   1:L PR[91] R[100]mm/sec CNT100;
   1:  PR[GP1:91,1] = PR[GP1:90,1] + -9.731;
   1:  PR[GP1:91,2] = PR[GP1:90,2] + -19.445;
   1:L PR[91] R[100]mm/sec CNT100;
   1:  PR[GP1:91,1] = PR[GP1:90,1] + -5.449;
   1:  PR[GP1:91,2] = PR[GP1:90,2] + -10.889;
   1:L PR[91] R[100]mm/sec CNT100;
   1:  PR[GP1:91,1] = PR[GP1:90,1] + -4.653;
   1:  PR[GP1:91,2] = PR[GP1:90,2] + -8.576;
   1:L PR[91] R[100]mm/sec CNT100;
   1:  PR[GP1:91,1] = PR[GP1:90,1] + -3.640;
   1:  PR[GP1:91,2] = PR[GP1:90,2] + -7.457;
   1:L PR[91] R[100]mm/sec CNT100;
   1:  PR[GP1:91,1] = PR[GP1:90,1] + -3.365;
   1:  PR[GP1:91,2] = PR[GP1:90,2] + -7.289;
   1:L PR[91] R[100]mm/sec CNT100;
   1:  PR[GP1:91,1] = PR[GP1:90,1] + -1.883;
   1:  PR[GP1:91,2] = PR[GP1:90,2] + -5.517;
   1:L PR[91] R[100]mm/sec CNT100;
   1:  PR[GP1:91,1] = PR[GP1:90,1] + 0.854;
   1:  PR[GP1:91,2] = PR[GP1:90,2] + -5.728;
   1:L PR[91] R[100]mm/sec CNT100;
   1:  PR[GP1:91,1] = PR[GP1:90,1] + 0.970;
   1:  PR[GP1:91,2] = PR[GP1:90,2] + -5.821;
   1:L PR[91] R[100]mm/sec CNT100;
   1:  PR[GP1:91,1] = PR[GP1:90,1] + 2.632;
   1:  PR[GP1:91,2] = PR[GP1:90,2] + -5.804;
   1:L PR[91] R[100]mm/sec CNT100;
   1:  PR[GP1:91,1] = PR[GP1:90,1] + 3.827;
   1:  PR[GP1:91,2] = PR[GP1:90,2] + -8.079;
   1:L PR[91] R[100]mm/sec CNT100;
   1:  PR[GP1:91,1] = PR[GP1:90,1] + 5.267;
   1:  PR[GP1:91,2] = PR[GP1:90,2] + -9.737;
   1:L PR[91] R[100]mm/sec CNT100;
   1:  PR[GP1:91,1] = PR[GP1:90,1] + 5.657;
   1:  PR[GP1:91,2] = PR[GP1:90,2] + -10.885;
   1:L PR[91] R[100]mm/sec CNT100;
   1:  PR[GP1:91,1] = PR[GP1:90,1] + 9.936;
   1:  PR[GP1:91,2] = PR[GP1:90,2] + -19.424;
   1:L PR[91] R[100]mm/sec CNT100;
   1:  PR[GP1:91,1] = PR[GP1:90,1] + 11.362;
   1:  PR[GP1:91,2] = PR[GP1:90,2] + -21.256;
   1:L PR[91] R[100]mm/sec CNT100;
   1:  PR[GP1:91,1] = PR[GP1:90,1] + 17.225;
   1:  PR[GP1:91,2] = PR[GP1:90,2] + -27.151;
   1:L PR[91] R[100]mm/sec CNT100;
   1:  PR[GP1:91,1] = PR[GP1:90,1] + 20.403;
   1:  PR[GP1:91,2] = PR[GP1:90,2] + -29.215;
   1:L PR[91] R[100]mm/sec CNT100;
   1:  PR[GP1:91,1] = PR[GP1:90,1] + 26.588;
   1:  PR[GP1:91,2] = PR[GP1:90,2] + -32.377;
   1:L PR[91] R[100]mm/sec CNT100;
   1:  PR[GP1:91,1] = PR[GP1:90,1] + 31.844;
   1:  PR[GP1:91,2] = PR[GP1:90,2] + -33.700;
   1:L PR[91] R[100]mm/sec CNT100;
   1:  PR[GP1:91,1] = PR[GP1:90,1] + 37.254;
   1:  PR[GP1:91,2] = PR[GP1:90,2] + -34.580;
   1:L PR[91] R[100]mm/sec CNT100;
   1:  PR[GP1:91,1] = PR[GP1:90,1] + 44.180;
   1:  PR[GP1:91,2] = PR[GP1:90,2] + -34.012;
   1:L PR[91] R[100]mm/sec CNT100;
   1:  PR[GP1:91,1] = PR[GP1:90,1] + 48.239;
   1:  PR[GP1:91,2] = PR[GP1:90,2] + -33.396;
   1:L PR[91] R[100]mm/sec CNT100;
   1:  PR[GP1:91,1] = PR[GP1:90,1] + 55.770;
   1:  PR[GP1:91,2] = PR[GP1:90,2] + -30.124;
   1:L PR[91] R[100]mm/sec CNT100;
   1:  PR[GP1:91,1] = PR[GP1:90,1] + 58.421;
   1:  PR[GP1:91,2] = PR[GP1:90,2] + -28.802;
   1:L PR[91] R[100]mm/sec CNT100;
   1:  PR[GP1:91,1] = PR[GP1:90,1] + 65.161;
   1:  PR[GP1:91,2] = PR[GP1:90,2] + -22.652;
   1:L PR[91] R[100]mm/sec CNT100;
   1:  PR[GP1:91,1] = PR[GP1:90,1] + 66.678;
   1:  PR[GP1:91,2] = PR[GP1:90,2] + -21.157;
   1:L PR[91] R[100]mm/sec CNT100;
   1:  PR[GP1:91,1] = PR[GP1:90,1] + 71.318;
   1:  PR[GP1:91,2] = PR[GP1:90,2] + -12.665;
   1:L PR[91] R[100]mm/sec CNT100;
   1:  PR[GP1:91,1] = PR[GP1:90,1] + 72.060;
   1:  PR[GP1:91,2] = PR[GP1:90,2] + -11.235;
   1:L PR[91] R[100]mm/sec CNT100;
   1:  PR[GP1:91,1] = PR[GP1:90,1] + 73.937;
   1:  PR[GP1:91,2] = PR[GP1:90,2] + -0.072;
   1:L PR[91] R[100]mm/sec CNT100;
   1:  PR[GP1:91,1] = PR[GP1:90,1] + 72.293;
   1:  PR[GP1:91,2] = PR[GP1:90,2] + 9.629;
   1:L PR[91] R[100]mm/sec CNT100;
   1:  PR[GP1:91,1] = PR[GP1:90,1] + 72.058;
   1:  PR[GP1:91,2] = PR[GP1:90,2] + 11.094;
   1:L PR[91] R[100]mm/sec CNT100;
   1:  PR[GP1:91,1] = PR[GP1:90,1] + 71.318;
   1:  PR[GP1:91,2] = PR[GP1:90,2] + 12.521;
   1:L PR[91] R[100]mm/sec CNT100;
   1:  PR[GP1:91,1] = PR[GP1:90,1] + 66.678;
   1:  PR[GP1:91,2] = PR[GP1:90,2] + 21.013;
   1:L PR[91] R[100]mm/sec CNT100;
   1:  PR[GP1:91,1] = PR[GP1:90,1] + 65.161;
   1:  PR[GP1:91,2] = PR[GP1:90,2] + 22.508;
   1:L PR[91] R[100]mm/sec CNT100;
   1:  PR[GP1:91,1] = PR[GP1:90,1] + 58.420;
   1:  PR[GP1:91,2] = PR[GP1:90,2] + 28.658;
   1:L PR[91] R[100]mm/sec CNT100;
   1:  PR[GP1:91,1] = PR[GP1:90,1] + 55.770;
   1:  PR[GP1:91,2] = PR[GP1:90,2] + 29.980;
   1:L PR[91] R[100]mm/sec CNT100;
   1:  PR[GP1:91,1] = PR[GP1:90,1] + 48.239;
   1:  PR[GP1:91,2] = PR[GP1:90,2] + 33.252;
   1:L PR[91] R[100]mm/sec CNT100;
   1:  PR[GP1:91,1] = PR[GP1:90,1] + 44.180;
   1:  PR[GP1:91,2] = PR[GP1:90,2] + 33.868;
   1:L PR[91] R[100]mm/sec CNT100;
   1:  PR[GP1:91,1] = PR[GP1:90,1] + 37.254;
   1:  PR[GP1:91,2] = PR[GP1:90,2] + 34.436;
   1:L PR[91] R[100]mm/sec CNT100;
   1:  PR[GP1:91,1] = PR[GP1:90,1] + 31.844;
   1:  PR[GP1:91,2] = PR[GP1:90,2] + 33.556;
   1:L PR[91] R[100]mm/sec CNT100;
   1:  PR[GP1:91,1] = PR[GP1:90,1] + 26.588;
   1:  PR[GP1:91,2] = PR[GP1:90,2] + 32.233;
   1:L PR[91] R[100]mm/sec CNT100;
   1:  PR[GP1:91,1] = PR[GP1:90,1] + 20.403;
   1:  PR[GP1:91,2] = PR[GP1:90,2] + 29.071;
   1:L PR[91] R[100]mm/sec CNT100;
   1:  PR[GP1:91,1] = PR[GP1:90,1] + 17.225;
   1:  PR[GP1:91,2] = PR[GP1:90,2] + 27.007;
   1:L PR[91] R[100]mm/sec CNT100;
   1:  PR[GP1:91,1] = PR[GP1:90,1] + 11.362;
   1:  PR[GP1:91,2] = PR[GP1:90,2] + 21.112;
   1:L PR[91] R[100]mm/sec CNT100;
   1:  PR[GP1:91,1] = PR[GP1:90,1] + 9.936;
   1:  PR[GP1:91,2] = PR[GP1:90,2] + 19.280;
   1:L PR[91] R[100]mm/sec CNT100;
   1:  PR[GP1:91,1] = PR[GP1:90,1] + 5.650;
   1:  PR[GP1:91,2] = PR[GP1:90,2] + 10.721;
   1:L PR[91] R[100]mm/sec CNT100;
   1:  PR[GP1:91,1] = PR[GP1:90,1] + 4.861;
   1:  PR[GP1:91,2] = PR[GP1:90,2] + 8.427;
   1:L PR[91] R[100]mm/sec CNT100;
   1:  PR[GP1:91,1] = PR[GP1:90,1] + 3.470;
   1:  PR[GP1:91,2] = PR[GP1:90,2] + 6.742;
   1:L PR[91] R[100]mm/sec CNT100;
   1:  PR[GP1:91,1] = PR[GP1:90,1] + 2.488;
   1:  PR[GP1:91,2] = PR[GP1:90,2] + 5.675;
   1:L PR[91] R[100]mm/sec CNT100;
   1:  PR[GP1:91,1] = PR[GP1:90,1] + 1.953;
   1:  PR[GP1:91,2] = PR[GP1:90,2] + 5.378;
   1:L PR[91] R[100]mm/sec CNT100;
   1:  PR[GP1:91,1] = PR[GP1:90,1] + 0.318;
   1:  PR[GP1:91,2] = PR[GP1:90,2] + 5.396;
   1:L PR[91] R[100]mm/sec CNT100;
   1:  ! -- Layer/Ebene 36 -- !;
   1:  PR[91] = PR[90];
   1:  PR[GP1:91,1] = PR[GP1:90,1] + -2.118;
   1:  PR[GP1:91,2] = PR[GP1:90,2] + 6.097;
   1:  PR[GP1:91,3] = PR[GP1:90,3] + 22.265;
   1:L PR[91] R[100]mm/sec CNT100;
   1:  PR[GP1:91,1] = PR[GP1:90,1] + -2.464;
   1:  PR[GP1:91,2] = PR[GP1:90,2] + 6.339;
   1:L PR[91] R[100]mm/sec CNT100;
   1:  PR[GP1:91,1] = PR[GP1:90,1] + -4.032;
   1:  PR[GP1:91,2] = PR[GP1:90,2] + 8.260;
   1:L PR[91] R[100]mm/sec CNT100;
   1:  PR[GP1:91,1] = PR[GP1:90,1] + -5.055;
   1:  PR[GP1:91,2] = PR[GP1:90,2] + 10.096;
   1:L PR[91] R[100]mm/sec CNT100;
   1:  PR[GP1:91,1] = PR[GP1:90,1] + -5.086;
   1:  PR[GP1:91,2] = PR[GP1:90,2] + 10.184;
   1:L PR[91] R[100]mm/sec CNT100;
   1:  PR[GP1:91,1] = PR[GP1:90,1] + -9.811;
   1:  PR[GP1:91,2] = PR[GP1:90,2] + 19.632;
   1:L PR[91] R[100]mm/sec CNT100;
   1:  PR[GP1:91,1] = PR[GP1:90,1] + -10.635;
   1:  PR[GP1:91,2] = PR[GP1:90,2] + 20.691;
   1:L PR[91] R[100]mm/sec CNT100;
   1:  PR[GP1:91,1] = PR[GP1:90,1] + -17.148;
   1:  PR[GP1:91,2] = PR[GP1:90,2] + 27.222;
   1:L PR[91] R[100]mm/sec CNT100;
   1:  PR[GP1:91,1] = PR[GP1:90,1] + -19.550;
   1:  PR[GP1:91,2] = PR[GP1:90,2] + 28.782;
   1:L PR[91] R[100]mm/sec CNT100;
   1:  PR[GP1:91,1] = PR[GP1:90,1] + -26.512;
   1:  PR[GP1:91,2] = PR[GP1:90,2] + 32.342;
   1:L PR[91] R[100]mm/sec CNT100;
   1:  PR[GP1:91,1] = PR[GP1:90,1] + -30.929;
   1:  PR[GP1:91,2] = PR[GP1:90,2] + 33.452;
   1:L PR[91] R[100]mm/sec CNT100;
   1:  PR[GP1:91,1] = PR[GP1:90,1] + -37.146;
   1:  PR[GP1:91,2] = PR[GP1:90,2] + 34.460;
   1:L PR[91] R[100]mm/sec CNT100;
   1:  PR[GP1:91,1] = PR[GP1:90,1] + -43.275;
   1:  PR[GP1:91,2] = PR[GP1:90,2] + 33.958;
   1:L PR[91] R[100]mm/sec CNT100;
   1:  PR[GP1:91,1] = PR[GP1:90,1] + -48.084;
   1:  PR[GP1:91,2] = PR[GP1:90,2] + 33.227;
   1:L PR[91] R[100]mm/sec CNT100;
   1:  PR[GP1:91,1] = PR[GP1:90,1] + -54.936;
   1:  PR[GP1:91,2] = PR[GP1:90,2] + 30.249;
   1:L PR[91] R[100]mm/sec CNT100;
   1:  PR[GP1:91,1] = PR[GP1:90,1] + -58.218;
   1:  PR[GP1:91,2] = PR[GP1:90,2] + 28.610;
   1:L PR[91] R[100]mm/sec CNT100;
   1:  PR[GP1:91,1] = PR[GP1:90,1] + -64.451;
   1:  PR[GP1:91,2] = PR[GP1:90,2] + 22.925;
   1:L PR[91] R[100]mm/sec CNT100;
   1:  PR[GP1:91,1] = PR[GP1:90,1] + -66.435;
   1:  PR[GP1:91,2] = PR[GP1:90,2] + 20.972;
   1:L PR[91] R[100]mm/sec CNT100;
   1:  PR[GP1:91,1] = PR[GP1:90,1] + -70.765;
   1:  PR[GP1:91,2] = PR[GP1:90,2] + 13.041;
   1:L PR[91] R[100]mm/sec CNT100;
   1:  PR[GP1:91,1] = PR[GP1:90,1] + -71.790;
   1:  PR[GP1:91,2] = PR[GP1:90,2] + 11.059;
   1:L PR[91] R[100]mm/sec CNT100;
   1:  PR[GP1:91,1] = PR[GP1:90,1] + -73.381;
   1:  PR[GP1:91,2] = PR[GP1:90,2] + 1.661;
   1:L PR[91] R[100]mm/sec CNT100;
   1:  PR[GP1:91,1] = PR[GP1:90,1] + -73.658;
   1:  PR[GP1:91,2] = PR[GP1:90,2] + -0.069;
   1:L PR[91] R[100]mm/sec CNT100;
   1:  PR[GP1:91,1] = PR[GP1:90,1] + -72.112;
   1:  PR[GP1:91,2] = PR[GP1:90,2] + -9.183;
   1:L PR[91] R[100]mm/sec CNT100;
   1:  PR[GP1:91,1] = PR[GP1:90,1] + -71.789;
   1:  PR[GP1:91,2] = PR[GP1:90,2] + -11.206;
   1:L PR[91] R[100]mm/sec CNT100;
   1:  PR[GP1:91,1] = PR[GP1:90,1] + -70.765;
   1:  PR[GP1:91,2] = PR[GP1:90,2] + -13.185;
   1:L PR[91] R[100]mm/sec CNT100;
   1:  PR[GP1:91,1] = PR[GP1:90,1] + -66.435;
   1:  PR[GP1:91,2] = PR[GP1:90,2] + -21.116;
   1:L PR[91] R[100]mm/sec CNT100;
   1:  PR[GP1:91,1] = PR[GP1:90,1] + -64.451;
   1:  PR[GP1:91,2] = PR[GP1:90,2] + -23.069;
   1:L PR[91] R[100]mm/sec CNT100;
   1:  PR[GP1:91,1] = PR[GP1:90,1] + -58.218;
   1:  PR[GP1:91,2] = PR[GP1:90,2] + -28.754;
   1:L PR[91] R[100]mm/sec CNT100;
   1:  PR[GP1:91,1] = PR[GP1:90,1] + -54.936;
   1:  PR[GP1:91,2] = PR[GP1:90,2] + -30.393;
   1:L PR[91] R[100]mm/sec CNT100;
   1:  PR[GP1:91,1] = PR[GP1:90,1] + -48.084;
   1:  PR[GP1:91,2] = PR[GP1:90,2] + -33.371;
   1:L PR[91] R[100]mm/sec CNT100;
   1:  PR[GP1:91,1] = PR[GP1:90,1] + -43.275;
   1:  PR[GP1:91,2] = PR[GP1:90,2] + -34.102;
   1:L PR[91] R[100]mm/sec CNT100;
   1:  PR[GP1:91,1] = PR[GP1:90,1] + -37.146;
   1:  PR[GP1:91,2] = PR[GP1:90,2] + -34.604;
   1:L PR[91] R[100]mm/sec CNT100;
   1:  PR[GP1:91,1] = PR[GP1:90,1] + -30.929;
   1:  PR[GP1:91,2] = PR[GP1:90,2] + -33.597;
   1:L PR[91] R[100]mm/sec CNT100;
   1:  PR[GP1:91,1] = PR[GP1:90,1] + -26.512;
   1:  PR[GP1:91,2] = PR[GP1:90,2] + -32.486;
   1:L PR[91] R[100]mm/sec CNT100;
   1:  PR[GP1:91,1] = PR[GP1:90,1] + -19.550;
   1:  PR[GP1:91,2] = PR[GP1:90,2] + -28.926;
   1:L PR[91] R[100]mm/sec CNT100;
   1:  PR[GP1:91,1] = PR[GP1:90,1] + -17.148;
   1:  PR[GP1:91,2] = PR[GP1:90,2] + -27.366;
   1:L PR[91] R[100]mm/sec CNT100;
   1:  PR[GP1:91,1] = PR[GP1:90,1] + -10.636;
   1:  PR[GP1:91,2] = PR[GP1:90,2] + -20.835;
   1:L PR[91] R[100]mm/sec CNT100;
   1:  PR[GP1:91,1] = PR[GP1:90,1] + -9.811;
   1:  PR[GP1:91,2] = PR[GP1:90,2] + -19.776;
   1:L PR[91] R[100]mm/sec CNT100;
   1:  PR[GP1:91,1] = PR[GP1:90,1] + -5.092;
   1:  PR[GP1:91,2] = PR[GP1:90,2] + -10.348;
   1:L PR[91] R[100]mm/sec CNT100;
   1:  PR[GP1:91,1] = PR[GP1:90,1] + -4.686;
   1:  PR[GP1:91,2] = PR[GP1:90,2] + -9.176;
   1:L PR[91] R[100]mm/sec CNT100;
   1:  PR[GP1:91,1] = PR[GP1:90,1] + -3.811;
   1:  PR[GP1:91,2] = PR[GP1:90,2] + -8.208;
   1:L PR[91] R[100]mm/sec CNT100;
   1:  PR[GP1:91,1] = PR[GP1:90,1] + -3.581;
   1:  PR[GP1:91,2] = PR[GP1:90,2] + -8.068;
   1:L PR[91] R[100]mm/sec CNT100;
   1:  PR[GP1:91,1] = PR[GP1:90,1] + -1.892;
   1:  PR[GP1:91,2] = PR[GP1:90,2] + -6.051;
   1:L PR[91] R[100]mm/sec CNT100;
   1:  PR[GP1:91,1] = PR[GP1:90,1] + 0.607;
   1:  PR[GP1:91,2] = PR[GP1:90,2] + -6.243;
   1:L PR[91] R[100]mm/sec CNT100;
   1:  PR[GP1:91,1] = PR[GP1:90,1] + 0.708;
   1:  PR[GP1:91,2] = PR[GP1:90,2] + -6.324;
   1:L PR[91] R[100]mm/sec CNT100;
   1:  PR[GP1:91,1] = PR[GP1:90,1] + 2.587;
   1:  PR[GP1:91,2] = PR[GP1:90,2] + -6.305;
   1:L PR[91] R[100]mm/sec CNT100;
   1:  PR[GP1:91,1] = PR[GP1:90,1] + 3.671;
   1:  PR[GP1:91,2] = PR[GP1:90,2] + -8.367;
   1:L PR[91] R[100]mm/sec CNT100;
   1:  PR[GP1:91,1] = PR[GP1:90,1] + 5.242;
   1:  PR[GP1:91,2] = PR[GP1:90,2] + -10.177;
   1:L PR[91] R[100]mm/sec CNT100;
   1:  PR[GP1:91,1] = PR[GP1:90,1] + 5.299;
   1:  PR[GP1:91,2] = PR[GP1:90,2] + -10.344;
   1:L PR[91] R[100]mm/sec CNT100;
   1:  PR[GP1:91,1] = PR[GP1:90,1] + 10.015;
   1:  PR[GP1:91,2] = PR[GP1:90,2] + -19.754;
   1:L PR[91] R[100]mm/sec CNT100;
   1:  PR[GP1:91,1] = PR[GP1:90,1] + 10.839;
   1:  PR[GP1:91,2] = PR[GP1:90,2] + -20.812;
   1:L PR[91] R[100]mm/sec CNT100;
   1:  PR[GP1:91,1] = PR[GP1:90,1] + 17.352;
   1:  PR[GP1:91,2] = PR[GP1:90,2] + -27.362;
   1:L PR[91] R[100]mm/sec CNT100;
   1:  PR[GP1:91,1] = PR[GP1:90,1] + 19.752;
   1:  PR[GP1:91,2] = PR[GP1:90,2] + -28.920;
   1:L PR[91] R[100]mm/sec CNT100;
   1:  PR[GP1:91,1] = PR[GP1:90,1] + 26.717;
   1:  PR[GP1:91,2] = PR[GP1:90,2] + -32.481;
   1:L PR[91] R[100]mm/sec CNT100;
   1:  PR[GP1:91,1] = PR[GP1:90,1] + 31.133;
   1:  PR[GP1:91,2] = PR[GP1:90,2] + -33.593;
   1:L PR[91] R[100]mm/sec CNT100;
   1:  PR[GP1:91,1] = PR[GP1:90,1] + 37.353;
   1:  PR[GP1:91,2] = PR[GP1:90,2] + -34.604;
   1:L PR[91] R[100]mm/sec CNT100;
   1:  PR[GP1:91,1] = PR[GP1:90,1] + 43.481;
   1:  PR[GP1:91,2] = PR[GP1:90,2] + -34.102;
   1:L PR[91] R[100]mm/sec CNT100;
   1:  PR[GP1:91,1] = PR[GP1:90,1] + 48.293;
   1:  PR[GP1:91,2] = PR[GP1:90,2] + -33.372;
   1:L PR[91] R[100]mm/sec CNT100;
   1:  PR[GP1:91,1] = PR[GP1:90,1] + 55.145;
   1:  PR[GP1:91,2] = PR[GP1:90,2] + -30.394;
   1:L PR[91] R[100]mm/sec CNT100;
   1:  PR[GP1:91,1] = PR[GP1:90,1] + 58.429;
   1:  PR[GP1:91,2] = PR[GP1:90,2] + -28.757;
   1:L PR[91] R[100]mm/sec CNT100;
   1:  PR[GP1:91,1] = PR[GP1:90,1] + 64.662;
   1:  PR[GP1:91,2] = PR[GP1:90,2] + -23.070;
   1:L PR[91] R[100]mm/sec CNT100;
   1:  PR[GP1:91,1] = PR[GP1:90,1] + 66.647;
   1:  PR[GP1:91,2] = PR[GP1:90,2] + -21.114;
   1:L PR[91] R[100]mm/sec CNT100;
   1:  PR[GP1:91,1] = PR[GP1:90,1] + 70.978;
   1:  PR[GP1:91,2] = PR[GP1:90,2] + -13.188;
   1:L PR[91] R[100]mm/sec CNT100;
   1:  PR[GP1:91,1] = PR[GP1:90,1] + 72.003;
   1:  PR[GP1:91,2] = PR[GP1:90,2] + -11.210;
   1:L PR[91] R[100]mm/sec CNT100;
   1:  PR[GP1:91,1] = PR[GP1:90,1] + 73.594;
   1:  PR[GP1:91,2] = PR[GP1:90,2] + -1.807;
   1:L PR[91] R[100]mm/sec CNT100;
   1:  PR[GP1:91,1] = PR[GP1:90,1] + 73.871;
   1:  PR[GP1:91,2] = PR[GP1:90,2] + -0.075;
   1:L PR[91] R[100]mm/sec CNT100;
   1:  PR[GP1:91,1] = PR[GP1:90,1] + 72.325;
   1:  PR[GP1:91,2] = PR[GP1:90,2] + 9.043;
   1:L PR[91] R[100]mm/sec CNT100;
   1:  PR[GP1:91,1] = PR[GP1:90,1] + 72.002;
   1:  PR[GP1:91,2] = PR[GP1:90,2] + 11.069;
   1:L PR[91] R[100]mm/sec CNT100;
   1:  PR[GP1:91,1] = PR[GP1:90,1] + 70.978;
   1:  PR[GP1:91,2] = PR[GP1:90,2] + 13.044;
   1:L PR[91] R[100]mm/sec CNT100;
   1:  PR[GP1:91,1] = PR[GP1:90,1] + 66.647;
   1:  PR[GP1:91,2] = PR[GP1:90,2] + 20.970;
   1:L PR[91] R[100]mm/sec CNT100;
   1:  PR[GP1:91,1] = PR[GP1:90,1] + 64.662;
   1:  PR[GP1:91,2] = PR[GP1:90,2] + 22.926;
   1:L PR[91] R[100]mm/sec CNT100;
   1:  PR[GP1:91,1] = PR[GP1:90,1] + 58.428;
   1:  PR[GP1:91,2] = PR[GP1:90,2] + 28.613;
   1:L PR[91] R[100]mm/sec CNT100;
   1:  PR[GP1:91,1] = PR[GP1:90,1] + 55.145;
   1:  PR[GP1:91,2] = PR[GP1:90,2] + 30.250;
   1:L PR[91] R[100]mm/sec CNT100;
   1:  PR[GP1:91,1] = PR[GP1:90,1] + 48.293;
   1:  PR[GP1:91,2] = PR[GP1:90,2] + 33.228;
   1:L PR[91] R[100]mm/sec CNT100;
   1:  PR[GP1:91,1] = PR[GP1:90,1] + 43.481;
   1:  PR[GP1:91,2] = PR[GP1:90,2] + 33.958;
   1:L PR[91] R[100]mm/sec CNT100;
   1:  PR[GP1:91,1] = PR[GP1:90,1] + 37.353;
   1:  PR[GP1:91,2] = PR[GP1:90,2] + 34.460;
   1:L PR[91] R[100]mm/sec CNT100;
   1:  PR[GP1:91,1] = PR[GP1:90,1] + 31.133;
   1:  PR[GP1:91,2] = PR[GP1:90,2] + 33.448;
   1:L PR[91] R[100]mm/sec CNT100;
   1:  PR[GP1:91,1] = PR[GP1:90,1] + 26.717;
   1:  PR[GP1:91,2] = PR[GP1:90,2] + 32.337;
   1:L PR[91] R[100]mm/sec CNT100;
   1:  PR[GP1:91,1] = PR[GP1:90,1] + 19.752;
   1:  PR[GP1:91,2] = PR[GP1:90,2] + 28.776;
   1:L PR[91] R[100]mm/sec CNT100;
   1:  PR[GP1:91,1] = PR[GP1:90,1] + 17.352;
   1:  PR[GP1:91,2] = PR[GP1:90,2] + 27.218;
   1:L PR[91] R[100]mm/sec CNT100;
   1:  PR[GP1:91,1] = PR[GP1:90,1] + 10.839;
   1:  PR[GP1:91,2] = PR[GP1:90,2] + 20.668;
   1:L PR[91] R[100]mm/sec CNT100;
   1:  PR[GP1:91,1] = PR[GP1:90,1] + 10.015;
   1:  PR[GP1:91,2] = PR[GP1:90,2] + 19.610;
   1:L PR[91] R[100]mm/sec CNT100;
   1:  PR[GP1:91,1] = PR[GP1:90,1] + 5.291;
   1:  PR[GP1:91,2] = PR[GP1:90,2] + 10.178;
   1:L PR[91] R[100]mm/sec CNT100;
   1:  PR[GP1:91,1] = PR[GP1:90,1] + 4.894;
   1:  PR[GP1:91,2] = PR[GP1:90,2] + 9.025;
   1:L PR[91] R[100]mm/sec CNT100;
   1:  PR[GP1:91,1] = PR[GP1:90,1] + 3.346;
   1:  PR[GP1:91,2] = PR[GP1:90,2] + 7.151;
   1:L PR[91] R[100]mm/sec CNT100;
   1:  PR[GP1:91,1] = PR[GP1:90,1] + 2.460;
   1:  PR[GP1:91,2] = PR[GP1:90,2] + 6.187;
   1:L PR[91] R[100]mm/sec CNT100;
   1:  PR[GP1:91,1] = PR[GP1:90,1] + 1.958;
   1:  PR[GP1:91,2] = PR[GP1:90,2] + 5.909;
   1:L PR[91] R[100]mm/sec CNT100;
   1:  PR[GP1:91,1] = PR[GP1:90,1] + 0.101;
   1:  PR[GP1:91,2] = PR[GP1:90,2] + 5.929;
   1:L PR[91] R[100]mm/sec CNT100;
   1:  ! -- Layer/Ebene 37 -- !;
   1:  PR[91] = PR[90];
   1:  PR[GP1:91,1] = PR[GP1:90,1] + -2.095;
   1:  PR[GP1:91,2] = PR[GP1:90,2] + 6.612;
   1:  PR[GP1:91,3] = PR[GP1:90,3] + 22.875;
   1:L PR[91] R[100]mm/sec CNT100;
   1:  PR[GP1:91,1] = PR[GP1:90,1] + -2.424;
   1:  PR[GP1:91,2] = PR[GP1:90,2] + 6.842;
   1:L PR[91] R[100]mm/sec CNT100;
   1:  PR[GP1:91,1] = PR[GP1:90,1] + -4.178;
   1:  PR[GP1:91,2] = PR[GP1:90,2] + 8.991;
   1:L PR[91] R[100]mm/sec CNT100;
   1:  PR[GP1:91,1] = PR[GP1:90,1] + -5.004;
   1:  PR[GP1:91,2] = PR[GP1:90,2] + 10.477;
   1:L PR[91] R[100]mm/sec CNT100;
   1:  PR[GP1:91,1] = PR[GP1:90,1] + -8.299;
   1:  PR[GP1:91,2] = PR[GP1:90,2] + 16.783;
   1:L PR[91] R[100]mm/sec CNT100;
   1:  PR[GP1:91,1] = PR[GP1:90,1] + -9.890;
   1:  PR[GP1:91,2] = PR[GP1:90,2] + 19.964;
   1:L PR[91] R[100]mm/sec CNT100;
   1:  PR[GP1:91,1] = PR[GP1:90,1] + -10.113;
   1:  PR[GP1:91,2] = PR[GP1:90,2] + 20.250;
   1:L PR[91] R[100]mm/sec CNT100;
   1:  PR[GP1:91,1] = PR[GP1:90,1] + -17.276;
   1:  PR[GP1:91,2] = PR[GP1:90,2] + 27.433;
   1:L PR[91] R[100]mm/sec CNT100;
   1:  PR[GP1:91,1] = PR[GP1:90,1] + -18.899;
   1:  PR[GP1:91,2] = PR[GP1:90,2] + 28.487;
   1:L PR[91] R[100]mm/sec CNT100;
   1:  PR[GP1:91,1] = PR[GP1:90,1] + -26.641;
   1:  PR[GP1:91,2] = PR[GP1:90,2] + 32.446;
   1:L PR[91] R[100]mm/sec CNT100;
   1:  PR[GP1:91,1] = PR[GP1:90,1] + -30.219;
   1:  PR[GP1:91,2] = PR[GP1:90,2] + 33.346;
   1:L PR[91] R[100]mm/sec CNT100;
   1:  PR[GP1:91,1] = PR[GP1:90,1] + -37.246;
   1:  PR[GP1:91,2] = PR[GP1:90,2] + 34.485;
   1:L PR[91] R[100]mm/sec CNT100;
   1:  PR[GP1:91,1] = PR[GP1:90,1] + -42.576;
   1:  PR[GP1:91,2] = PR[GP1:90,2] + 34.048;
   1:L PR[91] R[100]mm/sec CNT100;
   1:  PR[GP1:91,1] = PR[GP1:90,1] + -48.139;
   1:  PR[GP1:91,2] = PR[GP1:90,2] + 33.203;
   1:L PR[91] R[100]mm/sec CNT100;
   1:  PR[GP1:91,1] = PR[GP1:90,1] + -54.313;
   1:  PR[GP1:91,2] = PR[GP1:90,2] + 30.519;
   1:L PR[91] R[100]mm/sec CNT100;
   1:  PR[GP1:91,1] = PR[GP1:90,1] + -58.226;
   1:  PR[GP1:91,2] = PR[GP1:90,2] + 28.565;
   1:L PR[91] R[100]mm/sec CNT100;
   1:  PR[GP1:91,1] = PR[GP1:90,1] + -63.952;
   1:  PR[GP1:91,2] = PR[GP1:90,2] + 23.343;
   1:L PR[91] R[100]mm/sec CNT100;
   1:  PR[GP1:91,1] = PR[GP1:90,1] + -66.404;
   1:  PR[GP1:91,2] = PR[GP1:90,2] + 20.929;
   1:L PR[91] R[100]mm/sec CNT100;
   1:  PR[GP1:91,1] = PR[GP1:90,1] + -70.425;
   1:  PR[GP1:91,2] = PR[GP1:90,2] + 13.564;
   1:L PR[91] R[100]mm/sec CNT100;
   1:  PR[GP1:91,1] = PR[GP1:90,1] + -71.733;
   1:  PR[GP1:91,2] = PR[GP1:90,2] + 11.034;
   1:L PR[91] R[100]mm/sec CNT100;
   1:  PR[GP1:91,1] = PR[GP1:90,1] + -73.219;
   1:  PR[GP1:91,2] = PR[GP1:90,2] + 2.257;
   1:L PR[91] R[100]mm/sec CNT100;
   1:  PR[GP1:91,1] = PR[GP1:90,1] + -73.592;
   1:  PR[GP1:91,2] = PR[GP1:90,2] + -0.069;
   1:L PR[91] R[100]mm/sec CNT100;
   1:  PR[GP1:91,1] = PR[GP1:90,1] + -72.145;
   1:  PR[GP1:91,2] = PR[GP1:90,2] + -8.598;
   1:L PR[91] R[100]mm/sec CNT100;
   1:  PR[GP1:91,1] = PR[GP1:90,1] + -71.732;
   1:  PR[GP1:91,2] = PR[GP1:90,2] + -11.180;
   1:L PR[91] R[100]mm/sec CNT100;
   1:  PR[GP1:91,1] = PR[GP1:90,1] + -70.425;
   1:  PR[GP1:91,2] = PR[GP1:90,2] + -13.708;
   1:L PR[91] R[100]mm/sec CNT100;
   1:  PR[GP1:91,1] = PR[GP1:90,1] + -66.404;
   1:  PR[GP1:91,2] = PR[GP1:90,2] + -21.073;
   1:L PR[91] R[100]mm/sec CNT100;
   1:  PR[GP1:91,1] = PR[GP1:90,1] + -63.952;
   1:  PR[GP1:91,2] = PR[GP1:90,2] + -23.487;
   1:L PR[91] R[100]mm/sec CNT100;
   1:  PR[GP1:91,1] = PR[GP1:90,1] + -58.226;
   1:  PR[GP1:91,2] = PR[GP1:90,2] + -28.709;
   1:L PR[91] R[100]mm/sec CNT100;
   1:  PR[GP1:91,1] = PR[GP1:90,1] + -54.313;
   1:  PR[GP1:91,2] = PR[GP1:90,2] + -30.663;
   1:L PR[91] R[100]mm/sec CNT100;
   1:  PR[GP1:91,1] = PR[GP1:90,1] + -48.139;
   1:  PR[GP1:91,2] = PR[GP1:90,2] + -33.347;
   1:L PR[91] R[100]mm/sec CNT100;
   1:  PR[GP1:91,1] = PR[GP1:90,1] + -42.576;
   1:  PR[GP1:91,2] = PR[GP1:90,2] + -34.192;
   1:L PR[91] R[100]mm/sec CNT100;
   1:  PR[GP1:91,1] = PR[GP1:90,1] + -37.246;
   1:  PR[GP1:91,2] = PR[GP1:90,2] + -34.629;
   1:L PR[91] R[100]mm/sec CNT100;
   1:  PR[GP1:91,1] = PR[GP1:90,1] + -30.219;
   1:  PR[GP1:91,2] = PR[GP1:90,2] + -33.490;
   1:L PR[91] R[100]mm/sec CNT100;
   1:  PR[GP1:91,1] = PR[GP1:90,1] + -26.641;
   1:  PR[GP1:91,2] = PR[GP1:90,2] + -32.590;
   1:L PR[91] R[100]mm/sec CNT100;
   1:  PR[GP1:91,1] = PR[GP1:90,1] + -18.900;
   1:  PR[GP1:91,2] = PR[GP1:90,2] + -28.631;
   1:L PR[91] R[100]mm/sec CNT100;
   1:  PR[GP1:91,1] = PR[GP1:90,1] + -17.276;
   1:  PR[GP1:91,2] = PR[GP1:90,2] + -27.577;
   1:L PR[91] R[100]mm/sec CNT100;
   1:  PR[GP1:91,1] = PR[GP1:90,1] + -10.113;
   1:  PR[GP1:91,2] = PR[GP1:90,2] + -20.394;
   1:L PR[91] R[100]mm/sec CNT100;
   1:  PR[GP1:91,1] = PR[GP1:90,1] + -9.890;
   1:  PR[GP1:91,2] = PR[GP1:90,2] + -20.108;
   1:L PR[91] R[100]mm/sec CNT100;
   1:  PR[GP1:91,1] = PR[GP1:90,1] + -8.272;
   1:  PR[GP1:91,2] = PR[GP1:90,2] + -16.875;
   1:L PR[91] R[100]mm/sec CNT100;
   1:  PR[GP1:91,1] = PR[GP1:90,1] + -5.028;
   1:  PR[GP1:91,2] = PR[GP1:90,2] + -10.668;
   1:L PR[91] R[100]mm/sec CNT100;
   1:  PR[GP1:91,1] = PR[GP1:90,1] + -4.720;
   1:  PR[GP1:91,2] = PR[GP1:90,2] + -9.777;
   1:L PR[91] R[100]mm/sec CNT100;
   1:  PR[GP1:91,1] = PR[GP1:90,1] + -3.982;
   1:  PR[GP1:91,2] = PR[GP1:90,2] + -8.960;
   1:L PR[91] R[100]mm/sec CNT100;
   1:  PR[GP1:91,1] = PR[GP1:90,1] + -3.796;
   1:  PR[GP1:91,2] = PR[GP1:90,2] + -8.847;
   1:L PR[91] R[100]mm/sec CNT100;
   1:  PR[GP1:91,1] = PR[GP1:90,1] + -1.902;
   1:  PR[GP1:91,2] = PR[GP1:90,2] + -6.584;
   1:L PR[91] R[100]mm/sec CNT100;
   1:  PR[GP1:91,1] = PR[GP1:90,1] + 0.360;
   1:  PR[GP1:91,2] = PR[GP1:90,2] + -6.758;
   1:L PR[91] R[100]mm/sec CNT100;
   1:  PR[GP1:91,1] = PR[GP1:90,1] + 0.446;
   1:  PR[GP1:91,2] = PR[GP1:90,2] + -6.827;
   1:L PR[91] R[100]mm/sec CNT100;
   1:  PR[GP1:91,1] = PR[GP1:90,1] + 2.542;
   1:  PR[GP1:91,2] = PR[GP1:90,2] + -6.806;
   1:L PR[91] R[100]mm/sec CNT100;
   1:  PR[GP1:91,1] = PR[GP1:90,1] + 3.514;
   1:  PR[GP1:91,2] = PR[GP1:90,2] + -8.655;
   1:L PR[91] R[100]mm/sec CNT100;
   1:  PR[GP1:91,1] = PR[GP1:90,1] + 5.181;
   1:  PR[GP1:91,2] = PR[GP1:90,2] + -10.562;
   1:L PR[91] R[100]mm/sec CNT100;
   1:  PR[GP1:91,1] = PR[GP1:90,1] + 8.486;
   1:  PR[GP1:91,2] = PR[GP1:90,2] + -16.876;
   1:L PR[91] R[100]mm/sec CNT100;
   1:  PR[GP1:91,1] = PR[GP1:90,1] + 10.094;
   1:  PR[GP1:91,2] = PR[GP1:90,2] + -20.084;
   1:L PR[91] R[100]mm/sec CNT100;
   1:  PR[GP1:91,1] = PR[GP1:90,1] + 10.315;
   1:  PR[GP1:91,2] = PR[GP1:90,2] + -20.369;
   1:L PR[91] R[100]mm/sec CNT100;
   1:  PR[GP1:91,1] = PR[GP1:90,1] + 17.479;
   1:  PR[GP1:91,2] = PR[GP1:90,2] + -27.572;
   1:L PR[91] R[100]mm/sec CNT100;
   1:  PR[GP1:91,1] = PR[GP1:90,1] + 19.100;
   1:  PR[GP1:91,2] = PR[GP1:90,2] + -28.625;
   1:L PR[91] R[100]mm/sec CNT100;
   1:  PR[GP1:91,1] = PR[GP1:90,1] + 26.845;
   1:  PR[GP1:91,2] = PR[GP1:90,2] + -32.585;
   1:L PR[91] R[100]mm/sec CNT100;
   1:  PR[GP1:91,1] = PR[GP1:90,1] + 30.422;
   1:  PR[GP1:91,2] = PR[GP1:90,2] + -33.485;
   1:L PR[91] R[100]mm/sec CNT100;
   1:  PR[GP1:91,1] = PR[GP1:90,1] + 37.452;
   1:  PR[GP1:91,2] = PR[GP1:90,2] + -34.629;
   1:L PR[91] R[100]mm/sec CNT100;
   1:  PR[GP1:91,1] = PR[GP1:90,1] + 42.782;
   1:  PR[GP1:91,2] = PR[GP1:90,2] + -34.192;
   1:L PR[91] R[100]mm/sec CNT100;
   1:  PR[GP1:91,1] = PR[GP1:90,1] + 48.348;
   1:  PR[GP1:91,2] = PR[GP1:90,2] + -33.347;
   1:L PR[91] R[100]mm/sec CNT100;
   1:  PR[GP1:91,1] = PR[GP1:90,1] + 54.521;
   1:  PR[GP1:91,2] = PR[GP1:90,2] + -30.664;
   1:L PR[91] R[100]mm/sec CNT100;
   1:  PR[GP1:91,1] = PR[GP1:90,1] + 58.437;
   1:  PR[GP1:91,2] = PR[GP1:90,2] + -28.712;
   1:L PR[91] R[100]mm/sec CNT100;
   1:  PR[GP1:91,1] = PR[GP1:90,1] + 64.162;
   1:  PR[GP1:91,2] = PR[GP1:90,2] + -23.488;
   1:L PR[91] R[100]mm/sec CNT100;
   1:  PR[GP1:91,1] = PR[GP1:90,1] + 66.616;
   1:  PR[GP1:91,2] = PR[GP1:90,2] + -21.070;
   1:L PR[91] R[100]mm/sec CNT100;
   1:  PR[GP1:91,1] = PR[GP1:90,1] + 70.638;
   1:  PR[GP1:91,2] = PR[GP1:90,2] + -13.710;
   1:L PR[91] R[100]mm/sec CNT100;
   1:  PR[GP1:91,1] = PR[GP1:90,1] + 71.946;
   1:  PR[GP1:91,2] = PR[GP1:90,2] + -11.186;
   1:L PR[91] R[100]mm/sec CNT100;
   1:  PR[GP1:91,1] = PR[GP1:90,1] + 73.432;
   1:  PR[GP1:91,2] = PR[GP1:90,2] + -2.405;
   1:L PR[91] R[100]mm/sec CNT100;
   1:  PR[GP1:91,1] = PR[GP1:90,1] + 73.805;
   1:  PR[GP1:91,2] = PR[GP1:90,2] + -0.075;
   1:L PR[91] R[100]mm/sec CNT100;
   1:  PR[GP1:91,1] = PR[GP1:90,1] + 72.358;
   1:  PR[GP1:91,2] = PR[GP1:90,2] + 8.458;
   1:L PR[91] R[100]mm/sec CNT100;
   1:  PR[GP1:91,1] = PR[GP1:90,1] + 71.945;
   1:  PR[GP1:91,2] = PR[GP1:90,2] + 11.044;
   1:L PR[91] R[100]mm/sec CNT100;
   1:  PR[GP1:91,1] = PR[GP1:90,1] + 70.638;
   1:  PR[GP1:91,2] = PR[GP1:90,2] + 13.566;
   1:L PR[91] R[100]mm/sec CNT100;
   1:  PR[GP1:91,1] = PR[GP1:90,1] + 66.616;
   1:  PR[GP1:91,2] = PR[GP1:90,2] + 20.926;
   1:L PR[91] R[100]mm/sec CNT100;
   1:  PR[GP1:91,1] = PR[GP1:90,1] + 64.162;
   1:  PR[GP1:91,2] = PR[GP1:90,2] + 23.344;
   1:L PR[91] R[100]mm/sec CNT100;
   1:  PR[GP1:91,1] = PR[GP1:90,1] + 58.436;
   1:  PR[GP1:91,2] = PR[GP1:90,2] + 28.568;
   1:L PR[91] R[100]mm/sec CNT100;
   1:  PR[GP1:91,1] = PR[GP1:90,1] + 54.521;
   1:  PR[GP1:91,2] = PR[GP1:90,2] + 30.520;
   1:L PR[91] R[100]mm/sec CNT100;
   1:  PR[GP1:91,1] = PR[GP1:90,1] + 48.348;
   1:  PR[GP1:91,2] = PR[GP1:90,2] + 33.203;
   1:L PR[91] R[100]mm/sec CNT100;
   1:  PR[GP1:91,1] = PR[GP1:90,1] + 42.782;
   1:  PR[GP1:91,2] = PR[GP1:90,2] + 34.048;
   1:L PR[91] R[100]mm/sec CNT100;
   1:  PR[GP1:91,1] = PR[GP1:90,1] + 37.452;
   1:  PR[GP1:91,2] = PR[GP1:90,2] + 34.485;
   1:L PR[91] R[100]mm/sec CNT100;
   1:  PR[GP1:91,1] = PR[GP1:90,1] + 30.422;
   1:  PR[GP1:91,2] = PR[GP1:90,2] + 33.341;
   1:L PR[91] R[100]mm/sec CNT100;
   1:  PR[GP1:91,1] = PR[GP1:90,1] + 26.845;
   1:  PR[GP1:91,2] = PR[GP1:90,2] + 32.441;
   1:L PR[91] R[100]mm/sec CNT100;
   1:  PR[GP1:91,1] = PR[GP1:90,1] + 19.100;
   1:  PR[GP1:91,2] = PR[GP1:90,2] + 28.481;
   1:L PR[91] R[100]mm/sec CNT100;
   1:  PR[GP1:91,1] = PR[GP1:90,1] + 17.479;
   1:  PR[GP1:91,2] = PR[GP1:90,2] + 27.428;
   1:L PR[91] R[100]mm/sec CNT100;
   1:  PR[GP1:91,1] = PR[GP1:90,1] + 10.315;
   1:  PR[GP1:91,2] = PR[GP1:90,2] + 20.225;
   1:L PR[91] R[100]mm/sec CNT100;
   1:  PR[GP1:91,1] = PR[GP1:90,1] + 10.094;
   1:  PR[GP1:91,2] = PR[GP1:90,2] + 19.940;
   1:L PR[91] R[100]mm/sec CNT100;
   1:  PR[GP1:91,1] = PR[GP1:90,1] + 8.512;
   1:  PR[GP1:91,2] = PR[GP1:90,2] + 16.783;
   1:L PR[91] R[100]mm/sec CNT100;
   1:  PR[GP1:91,1] = PR[GP1:90,1] + 5.235;
   1:  PR[GP1:91,2] = PR[GP1:90,2] + 10.521;
   1:L PR[91] R[100]mm/sec CNT100;
   1:  PR[GP1:91,1] = PR[GP1:90,1] + 4.927;
   1:  PR[GP1:91,2] = PR[GP1:90,2] + 9.623;
   1:L PR[91] R[100]mm/sec CNT100;
   1:  PR[GP1:91,1] = PR[GP1:90,1] + 3.223;
   1:  PR[GP1:91,2] = PR[GP1:90,2] + 7.560;
   1:L PR[91] R[100]mm/sec CNT100;
   1:  PR[GP1:91,1] = PR[GP1:90,1] + 2.432;
   1:  PR[GP1:91,2] = PR[GP1:90,2] + 6.700;
   1:L PR[91] R[100]mm/sec CNT100;
   1:  PR[GP1:91,1] = PR[GP1:90,1] + 1.963;
   1:  PR[GP1:91,2] = PR[GP1:90,2] + 6.440;
   1:L PR[91] R[100]mm/sec CNT100;
   1:  PR[GP1:91,1] = PR[GP1:90,1] + -0.117;
   1:  PR[GP1:91,2] = PR[GP1:90,2] + 6.462;
   1:L PR[91] R[100]mm/sec CNT100;
   1:  ! -- Layer/Ebene 38 -- !;
   1:  PR[91] = PR[90];
   1:  PR[GP1:91,1] = PR[GP1:90,1] + -2.072;
   1:  PR[GP1:91,2] = PR[GP1:90,2] + 7.127;
   1:  PR[GP1:91,3] = PR[GP1:90,3] + 23.485;
   1:L PR[91] R[100]mm/sec CNT100;
   1:  PR[GP1:91,1] = PR[GP1:90,1] + -2.384;
   1:  PR[GP1:91,2] = PR[GP1:90,2] + 7.345;
   1:L PR[91] R[100]mm/sec CNT100;
   1:  PR[GP1:91,1] = PR[GP1:90,1] + -4.324;
   1:  PR[GP1:91,2] = PR[GP1:90,2] + 9.722;
   1:L PR[91] R[100]mm/sec CNT100;
   1:  PR[GP1:91,1] = PR[GP1:90,1] + -4.974;
   1:  PR[GP1:91,2] = PR[GP1:90,2] + 10.891;
   1:L PR[91] R[100]mm/sec CNT100;
   1:  PR[GP1:91,1] = PR[GP1:90,1] + -9.660;
   1:  PR[GP1:91,2] = PR[GP1:90,2] + 19.858;
   1:L PR[91] R[100]mm/sec CNT100;
   1:  PR[GP1:91,1] = PR[GP1:90,1] + -9.901;
   1:  PR[GP1:91,2] = PR[GP1:90,2] + 20.206;
   1:L PR[91] R[100]mm/sec CNT100;
   1:  PR[GP1:91,1] = PR[GP1:90,1] + -12.238;
   1:  PR[GP1:91,2] = PR[GP1:90,2] + 22.464;
   1:L PR[91] R[100]mm/sec CNT100;
   1:  PR[GP1:91,1] = PR[GP1:90,1] + -17.403;
   1:  PR[GP1:91,2] = PR[GP1:90,2] + 27.644;
   1:L PR[91] R[100]mm/sec CNT100;
   1:  PR[GP1:91,1] = PR[GP1:90,1] + -18.249;
   1:  PR[GP1:91,2] = PR[GP1:90,2] + 28.193;
   1:L PR[91] R[100]mm/sec CNT100;
   1:  PR[GP1:91,1] = PR[GP1:90,1] + -26.770;
   1:  PR[GP1:91,2] = PR[GP1:90,2] + 32.550;
   1:L PR[91] R[100]mm/sec CNT100;
   1:  PR[GP1:91,1] = PR[GP1:90,1] + -29.509;
   1:  PR[GP1:91,2] = PR[GP1:90,2] + 33.239;
   1:L PR[91] R[100]mm/sec CNT100;
   1:  PR[GP1:91,1] = PR[GP1:90,1] + -37.345;
   1:  PR[GP1:91,2] = PR[GP1:90,2] + 34.509;
   1:L PR[91] R[100]mm/sec CNT100;
   1:  PR[GP1:91,1] = PR[GP1:90,1] + -41.878;
   1:  PR[GP1:91,2] = PR[GP1:90,2] + 34.137;
   1:L PR[91] R[100]mm/sec CNT100;
   1:  PR[GP1:91,1] = PR[GP1:90,1] + -48.194;
   1:  PR[GP1:91,2] = PR[GP1:90,2] + 33.178;
   1:L PR[91] R[100]mm/sec CNT100;
   1:  PR[GP1:91,1] = PR[GP1:90,1] + -53.689;
   1:  PR[GP1:91,2] = PR[GP1:90,2] + 30.789;
   1:L PR[91] R[100]mm/sec CNT100;
   1:  PR[GP1:91,1] = PR[GP1:90,1] + -58.234;
   1:  PR[GP1:91,2] = PR[GP1:90,2] + 28.520;
   1:L PR[91] R[100]mm/sec CNT100;
   1:  PR[GP1:91,1] = PR[GP1:90,1] + -63.452;
   1:  PR[GP1:91,2] = PR[GP1:90,2] + 23.760;
   1:L PR[91] R[100]mm/sec CNT100;
   1:  PR[GP1:91,1] = PR[GP1:90,1] + -66.373;
   1:  PR[GP1:91,2] = PR[GP1:90,2] + 20.886;
   1:L PR[91] R[100]mm/sec CNT100;
   1:  PR[GP1:91,1] = PR[GP1:90,1] + -70.085;
   1:  PR[GP1:91,2] = PR[GP1:90,2] + 14.087;
   1:L PR[91] R[100]mm/sec CNT100;
   1:  PR[GP1:91,1] = PR[GP1:90,1] + -71.676;
   1:  PR[GP1:91,2] = PR[GP1:90,2] + 11.009;
   1:L PR[91] R[100]mm/sec CNT100;
   1:  PR[GP1:91,1] = PR[GP1:90,1] + -73.057;
   1:  PR[GP1:91,2] = PR[GP1:90,2] + 2.853;
   1:L PR[91] R[100]mm/sec CNT100;
   1:  PR[GP1:91,1] = PR[GP1:90,1] + -73.525;
   1:  PR[GP1:91,2] = PR[GP1:90,2] + -0.069;
   1:L PR[91] R[100]mm/sec CNT100;
   1:  PR[GP1:91,1] = PR[GP1:90,1] + -72.178;
   1:  PR[GP1:91,2] = PR[GP1:90,2] + -8.013;
   1:L PR[91] R[100]mm/sec CNT100;
   1:  PR[GP1:91,1] = PR[GP1:90,1] + -71.675;
   1:  PR[GP1:91,2] = PR[GP1:90,2] + -11.155;
   1:L PR[91] R[100]mm/sec CNT100;
   1:  PR[GP1:91,1] = PR[GP1:90,1] + -70.085;
   1:  PR[GP1:91,2] = PR[GP1:90,2] + -14.231;
   1:L PR[91] R[100]mm/sec CNT100;
   1:  PR[GP1:91,1] = PR[GP1:90,1] + -66.373;
   1:  PR[GP1:91,2] = PR[GP1:90,2] + -21.030;
   1:L PR[91] R[100]mm/sec CNT100;
   1:  PR[GP1:91,1] = PR[GP1:90,1] + -63.452;
   1:  PR[GP1:91,2] = PR[GP1:90,2] + -23.904;
   1:L PR[91] R[100]mm/sec CNT100;
   1:  PR[GP1:91,1] = PR[GP1:90,1] + -58.234;
   1:  PR[GP1:91,2] = PR[GP1:90,2] + -28.663;
   1:L PR[91] R[100]mm/sec CNT100;
   1:  PR[GP1:91,1] = PR[GP1:90,1] + -53.689;
   1:  PR[GP1:91,2] = PR[GP1:90,2] + -30.933;
   1:L PR[91] R[100]mm/sec CNT100;
   1:  PR[GP1:91,1] = PR[GP1:90,1] + -48.194;
   1:  PR[GP1:91,2] = PR[GP1:90,2] + -33.322;
   1:L PR[91] R[100]mm/sec CNT100;
   1:  PR[GP1:91,1] = PR[GP1:90,1] + -41.878;
   1:  PR[GP1:91,2] = PR[GP1:90,2] + -34.281;
   1:L PR[91] R[100]mm/sec CNT100;
   1:  PR[GP1:91,1] = PR[GP1:90,1] + -37.345;
   1:  PR[GP1:91,2] = PR[GP1:90,2] + -34.653;
   1:L PR[91] R[100]mm/sec CNT100;
   1:  PR[GP1:91,1] = PR[GP1:90,1] + -29.509;
   1:  PR[GP1:91,2] = PR[GP1:90,2] + -33.383;
   1:L PR[91] R[100]mm/sec CNT100;
   1:  PR[GP1:91,1] = PR[GP1:90,1] + -26.770;
   1:  PR[GP1:91,2] = PR[GP1:90,2] + -32.694;
   1:L PR[91] R[100]mm/sec CNT100;
   1:  PR[GP1:91,1] = PR[GP1:90,1] + -18.249;
   1:  PR[GP1:91,2] = PR[GP1:90,2] + -28.337;
   1:L PR[91] R[100]mm/sec CNT100;
   1:  PR[GP1:91,1] = PR[GP1:90,1] + -17.403;
   1:  PR[GP1:91,2] = PR[GP1:90,2] + -27.788;
   1:L PR[91] R[100]mm/sec CNT100;
   1:  PR[GP1:91,1] = PR[GP1:90,1] + -12.238;
   1:  PR[GP1:91,2] = PR[GP1:90,2] + -22.607;
   1:L PR[91] R[100]mm/sec CNT100;
   1:  PR[GP1:91,1] = PR[GP1:90,1] + -9.901;
   1:  PR[GP1:91,2] = PR[GP1:90,2] + -20.351;
   1:L PR[91] R[100]mm/sec CNT100;
   1:  PR[GP1:91,1] = PR[GP1:90,1] + -9.659;
   1:  PR[GP1:91,2] = PR[GP1:90,2] + -20.000;
   1:L PR[91] R[100]mm/sec CNT100;
   1:  PR[GP1:91,1] = PR[GP1:90,1] + -4.998;
   1:  PR[GP1:91,2] = PR[GP1:90,2] + -11.082;
   1:L PR[91] R[100]mm/sec CNT100;
   1:  PR[GP1:91,1] = PR[GP1:90,1] + -4.754;
   1:  PR[GP1:91,2] = PR[GP1:90,2] + -10.377;
   1:L PR[91] R[100]mm/sec CNT100;
   1:  PR[GP1:91,1] = PR[GP1:90,1] + -4.153;
   1:  PR[GP1:91,2] = PR[GP1:90,2] + -9.712;
   1:L PR[91] R[100]mm/sec CNT100;
   1:  PR[GP1:91,1] = PR[GP1:90,1] + -4.012;
   1:  PR[GP1:91,2] = PR[GP1:90,2] + -9.626;
   1:L PR[91] R[100]mm/sec CNT100;
   1:  PR[GP1:91,1] = PR[GP1:90,1] + -1.912;
   1:  PR[GP1:91,2] = PR[GP1:90,2] + -7.117;
   1:L PR[91] R[100]mm/sec CNT100;
   1:  PR[GP1:91,1] = PR[GP1:90,1] + 0.114;
   1:  PR[GP1:91,2] = PR[GP1:90,2] + -7.273;
   1:L PR[91] R[100]mm/sec CNT100;
   1:  PR[GP1:91,1] = PR[GP1:90,1] + 0.185;
   1:  PR[GP1:91,2] = PR[GP1:90,2] + -7.330;
   1:L PR[91] R[100]mm/sec CNT100;
   1:  PR[GP1:91,1] = PR[GP1:90,1] + 2.498;
   1:  PR[GP1:91,2] = PR[GP1:90,2] + -7.307;
   1:L PR[91] R[100]mm/sec CNT100;
   1:  PR[GP1:91,1] = PR[GP1:90,1] + 3.358;
   1:  PR[GP1:91,2] = PR[GP1:90,2] + -8.945;
   1:L PR[91] R[100]mm/sec CNT100;
   1:  PR[GP1:91,1] = PR[GP1:90,1] + 4.508;
   1:  PR[GP1:91,2] = PR[GP1:90,2] + -10.269;
   1:L PR[91] R[100]mm/sec CNT100;
   1:  PR[GP1:91,1] = PR[GP1:90,1] + 5.147;
   1:  PR[GP1:91,2] = PR[GP1:90,2] + -10.969;
   1:L PR[91] R[100]mm/sec CNT100;
   1:  PR[GP1:91,1] = PR[GP1:90,1] + 9.861;
   1:  PR[GP1:91,2] = PR[GP1:90,2] + -19.974;
   1:L PR[91] R[100]mm/sec CNT100;
   1:  PR[GP1:91,1] = PR[GP1:90,1] + 10.105;
   1:  PR[GP1:91,2] = PR[GP1:90,2] + -20.327;
   1:L PR[91] R[100]mm/sec CNT100;
   1:  PR[GP1:91,1] = PR[GP1:90,1] + 12.451;
   1:  PR[GP1:91,2] = PR[GP1:90,2] + -22.600;
   1:L PR[91] R[100]mm/sec CNT100;
   1:  PR[GP1:91,1] = PR[GP1:90,1] + 17.606;
   1:  PR[GP1:91,2] = PR[GP1:90,2] + -27.783;
   1:L PR[91] R[100]mm/sec CNT100;
   1:  PR[GP1:91,1] = PR[GP1:90,1] + 18.449;
   1:  PR[GP1:91,2] = PR[GP1:90,2] + -28.331;
   1:L PR[91] R[100]mm/sec CNT100;
   1:  PR[GP1:91,1] = PR[GP1:90,1] + 26.974;
   1:  PR[GP1:91,2] = PR[GP1:90,2] + -32.689;
   1:L PR[91] R[100]mm/sec CNT100;
   1:  PR[GP1:91,1] = PR[GP1:90,1] + 29.711;
   1:  PR[GP1:91,2] = PR[GP1:90,2] + -33.378;
   1:L PR[91] R[100]mm/sec CNT100;
   1:  PR[GP1:91,1] = PR[GP1:90,1] + 37.551;
   1:  PR[GP1:91,2] = PR[GP1:90,2] + -34.653;
   1:L PR[91] R[100]mm/sec CNT100;
   1:  PR[GP1:91,1] = PR[GP1:90,1] + 42.082;
   1:  PR[GP1:91,2] = PR[GP1:90,2] + -34.282;
   1:L PR[91] R[100]mm/sec CNT100;
   1:  PR[GP1:91,1] = PR[GP1:90,1] + 48.402;
   1:  PR[GP1:91,2] = PR[GP1:90,2] + -33.322;
   1:L PR[91] R[100]mm/sec CNT100;
   1:  PR[GP1:91,1] = PR[GP1:90,1] + 53.897;
   1:  PR[GP1:91,2] = PR[GP1:90,2] + -30.935;
   1:L PR[91] R[100]mm/sec CNT100;
   1:  PR[GP1:91,1] = PR[GP1:90,1] + 58.444;
   1:  PR[GP1:91,2] = PR[GP1:90,2] + -28.667;
   1:L PR[91] R[100]mm/sec CNT100;
   1:  PR[GP1:91,1] = PR[GP1:90,1] + 63.662;
   1:  PR[GP1:91,2] = PR[GP1:90,2] + -23.907;
   1:L PR[91] R[100]mm/sec CNT100;
   1:  PR[GP1:91,1] = PR[GP1:90,1] + 66.585;
   1:  PR[GP1:91,2] = PR[GP1:90,2] + -21.027;
   1:L PR[91] R[100]mm/sec CNT100;
   1:  PR[GP1:91,1] = PR[GP1:90,1] + 70.297;
   1:  PR[GP1:91,2] = PR[GP1:90,2] + -14.233;
   1:L PR[91] R[100]mm/sec CNT100;
   1:  PR[GP1:91,1] = PR[GP1:90,1] + 71.889;
   1:  PR[GP1:91,2] = PR[GP1:90,2] + -11.161;
   1:L PR[91] R[100]mm/sec CNT100;
   1:  PR[GP1:91,1] = PR[GP1:90,1] + 73.270;
   1:  PR[GP1:91,2] = PR[GP1:90,2] + -3.002;
   1:L PR[91] R[100]mm/sec CNT100;
   1:  PR[GP1:91,1] = PR[GP1:90,1] + 73.738;
   1:  PR[GP1:91,2] = PR[GP1:90,2] + -0.075;
   1:L PR[91] R[100]mm/sec CNT100;
   1:  PR[GP1:91,1] = PR[GP1:90,1] + 72.391;
   1:  PR[GP1:91,2] = PR[GP1:90,2] + 7.873;
   1:L PR[91] R[100]mm/sec CNT100;
   1:  PR[GP1:91,1] = PR[GP1:90,1] + 71.888;
   1:  PR[GP1:91,2] = PR[GP1:90,2] + 11.020;
   1:L PR[91] R[100]mm/sec CNT100;
   1:  PR[GP1:91,1] = PR[GP1:90,1] + 70.297;
   1:  PR[GP1:91,2] = PR[GP1:90,2] + 14.089;
   1:L PR[91] R[100]mm/sec CNT100;
   1:  PR[GP1:91,1] = PR[GP1:90,1] + 66.585;
   1:  PR[GP1:91,2] = PR[GP1:90,2] + 20.883;
   1:L PR[91] R[100]mm/sec CNT100;
   1:  PR[GP1:91,1] = PR[GP1:90,1] + 63.663;
   1:  PR[GP1:91,2] = PR[GP1:90,2] + 23.762;
   1:L PR[91] R[100]mm/sec CNT100;
   1:  PR[GP1:91,1] = PR[GP1:90,1] + 58.444;
   1:  PR[GP1:91,2] = PR[GP1:90,2] + 28.523;
   1:L PR[91] R[100]mm/sec CNT100;
   1:  PR[GP1:91,1] = PR[GP1:90,1] + 53.897;
   1:  PR[GP1:91,2] = PR[GP1:90,2] + 30.791;
   1:L PR[91] R[100]mm/sec CNT100;
   1:  PR[GP1:91,1] = PR[GP1:90,1] + 48.402;
   1:  PR[GP1:91,2] = PR[GP1:90,2] + 33.178;
   1:L PR[91] R[100]mm/sec CNT100;
   1:  PR[GP1:91,1] = PR[GP1:90,1] + 42.082;
   1:  PR[GP1:91,2] = PR[GP1:90,2] + 34.138;
   1:L PR[91] R[100]mm/sec CNT100;
   1:  PR[GP1:91,1] = PR[GP1:90,1] + 37.551;
   1:  PR[GP1:91,2] = PR[GP1:90,2] + 34.509;
   1:L PR[91] R[100]mm/sec CNT100;
   1:  PR[GP1:91,1] = PR[GP1:90,1] + 29.710;
   1:  PR[GP1:91,2] = PR[GP1:90,2] + 33.234;
   1:L PR[91] R[100]mm/sec CNT100;
   1:  PR[GP1:91,1] = PR[GP1:90,1] + 26.973;
   1:  PR[GP1:91,2] = PR[GP1:90,2] + 32.545;
   1:L PR[91] R[100]mm/sec CNT100;
   1:  PR[GP1:91,1] = PR[GP1:90,1] + 18.449;
   1:  PR[GP1:91,2] = PR[GP1:90,2] + 28.187;
   1:L PR[91] R[100]mm/sec CNT100;
   1:  PR[GP1:91,1] = PR[GP1:90,1] + 17.606;
   1:  PR[GP1:91,2] = PR[GP1:90,2] + 27.639;
   1:L PR[91] R[100]mm/sec CNT100;
   1:  PR[GP1:91,1] = PR[GP1:90,1] + 12.452;
   1:  PR[GP1:91,2] = PR[GP1:90,2] + 22.456;
   1:L PR[91] R[100]mm/sec CNT100;
   1:  PR[GP1:91,1] = PR[GP1:90,1] + 10.104;
   1:  PR[GP1:91,2] = PR[GP1:90,2] + 20.183;
   1:L PR[91] R[100]mm/sec CNT100;
   1:  PR[GP1:91,1] = PR[GP1:90,1] + 9.862;
   1:  PR[GP1:91,2] = PR[GP1:90,2] + 19.832;
   1:L PR[91] R[100]mm/sec CNT100;
   1:  PR[GP1:91,1] = PR[GP1:90,1] + 5.204;
   1:  PR[GP1:91,2] = PR[GP1:90,2] + 10.935;
   1:L PR[91] R[100]mm/sec CNT100;
   1:  PR[GP1:91,1] = PR[GP1:90,1] + 4.959;
   1:  PR[GP1:91,2] = PR[GP1:90,2] + 10.221;
   1:L PR[91] R[100]mm/sec CNT100;
   1:  PR[GP1:91,1] = PR[GP1:90,1] + 3.100;
   1:  PR[GP1:91,2] = PR[GP1:90,2] + 7.969;
   1:L PR[91] R[100]mm/sec CNT100;
   1:  PR[GP1:91,1] = PR[GP1:90,1] + 2.404;
   1:  PR[GP1:91,2] = PR[GP1:90,2] + 7.212;
   1:L PR[91] R[100]mm/sec CNT100;
   1:  PR[GP1:91,1] = PR[GP1:90,1] + 1.968;
   1:  PR[GP1:91,2] = PR[GP1:90,2] + 6.971;
   1:L PR[91] R[100]mm/sec CNT100;
   1:  PR[GP1:91,1] = PR[GP1:90,1] + -0.335;
   1:  PR[GP1:91,2] = PR[GP1:90,2] + 6.995;
   1:L PR[91] R[100]mm/sec CNT100;
   1:  ! -- Layer/Ebene 39 -- !;
   1:  PR[91] = PR[90];
   1:  PR[GP1:91,1] = PR[GP1:90,1] + -2.049;
   1:  PR[GP1:91,2] = PR[GP1:90,2] + 7.641;
   1:  PR[GP1:91,3] = PR[GP1:90,3] + 24.095;
   1:L PR[91] R[100]mm/sec CNT100;
   1:  PR[GP1:91,1] = PR[GP1:90,1] + -2.344;
   1:  PR[GP1:91,2] = PR[GP1:90,2] + 7.848;
   1:L PR[91] R[100]mm/sec CNT100;
   1:  PR[GP1:91,1] = PR[GP1:90,1] + -4.470;
   1:  PR[GP1:91,2] = PR[GP1:90,2] + 10.453;
   1:L PR[91] R[100]mm/sec CNT100;
   1:  PR[GP1:91,1] = PR[GP1:90,1] + -4.943;
   1:  PR[GP1:91,2] = PR[GP1:90,2] + 11.304;
   1:L PR[91] R[100]mm/sec CNT100;
   1:  PR[GP1:91,1] = PR[GP1:90,1] + -9.149;
   1:  PR[GP1:91,2] = PR[GP1:90,2] + 19.346;
   1:L PR[91] R[100]mm/sec CNT100;
   1:  PR[GP1:91,1] = PR[GP1:90,1] + -9.945;
   1:  PR[GP1:91,2] = PR[GP1:90,2] + 20.499;
   1:L PR[91] R[100]mm/sec CNT100;
   1:  PR[GP1:91,1] = PR[GP1:90,1] + -16.743;
   1:  PR[GP1:91,2] = PR[GP1:90,2] + 27.064;
   1:L PR[91] R[100]mm/sec CNT100;
   1:  PR[GP1:91,1] = PR[GP1:90,1] + -17.531;
   1:  PR[GP1:91,2] = PR[GP1:90,2] + 27.855;
   1:L PR[91] R[100]mm/sec CNT100;
   1:  PR[GP1:91,1] = PR[GP1:90,1] + -17.599;
   1:  PR[GP1:91,2] = PR[GP1:90,2] + 27.899;
   1:L PR[91] R[100]mm/sec CNT100;
   1:  PR[GP1:91,1] = PR[GP1:90,1] + -26.899;
   1:  PR[GP1:91,2] = PR[GP1:90,2] + 32.654;
   1:L PR[91] R[100]mm/sec CNT100;
   1:  PR[GP1:91,1] = PR[GP1:90,1] + -28.798;
   1:  PR[GP1:91,2] = PR[GP1:90,2] + 33.132;
   1:L PR[91] R[100]mm/sec CNT100;
   1:  PR[GP1:91,1] = PR[GP1:90,1] + -37.445;
   1:  PR[GP1:91,2] = PR[GP1:90,2] + 34.533;
   1:L PR[91] R[100]mm/sec CNT100;
   1:  PR[GP1:91,1] = PR[GP1:90,1] + -41.179;
   1:  PR[GP1:91,2] = PR[GP1:90,2] + 34.227;
   1:L PR[91] R[100]mm/sec CNT100;
   1:  PR[GP1:91,1] = PR[GP1:90,1] + -48.249;
   1:  PR[GP1:91,2] = PR[GP1:90,2] + 33.153;
   1:L PR[91] R[100]mm/sec CNT100;
   1:  PR[GP1:91,1] = PR[GP1:90,1] + -53.066;
   1:  PR[GP1:91,2] = PR[GP1:90,2] + 31.060;
   1:L PR[91] R[100]mm/sec CNT100;
   1:  PR[GP1:91,1] = PR[GP1:90,1] + -58.242;
   1:  PR[GP1:91,2] = PR[GP1:90,2] + 28.474;
   1:L PR[91] R[100]mm/sec CNT100;
   1:  PR[GP1:91,1] = PR[GP1:90,1] + -62.953;
   1:  PR[GP1:91,2] = PR[GP1:90,2] + 24.178;
   1:L PR[91] R[100]mm/sec CNT100;
   1:  PR[GP1:91,1] = PR[GP1:90,1] + -66.342;
   1:  PR[GP1:91,2] = PR[GP1:90,2] + 20.843;
   1:L PR[91] R[100]mm/sec CNT100;
   1:  PR[GP1:91,1] = PR[GP1:90,1] + -69.745;
   1:  PR[GP1:91,2] = PR[GP1:90,2] + 14.610;
   1:L PR[91] R[100]mm/sec CNT100;
   1:  PR[GP1:91,1] = PR[GP1:90,1] + -71.619;
   1:  PR[GP1:91,2] = PR[GP1:90,2] + 10.983;
   1:L PR[91] R[100]mm/sec CNT100;
   1:  PR[GP1:91,1] = PR[GP1:90,1] + -72.895;
   1:  PR[GP1:91,2] = PR[GP1:90,2] + 3.450;
   1:L PR[91] R[100]mm/sec CNT100;
   1:  PR[GP1:91,1] = PR[GP1:90,1] + -73.459;
   1:  PR[GP1:91,2] = PR[GP1:90,2] + -0.069;
   1:L PR[91] R[100]mm/sec CNT100;
   1:  PR[GP1:91,1] = PR[GP1:90,1] + -72.211;
   1:  PR[GP1:91,2] = PR[GP1:90,2] + -7.428;
   1:L PR[91] R[100]mm/sec CNT100;
   1:  PR[GP1:91,1] = PR[GP1:90,1] + -71.618;
   1:  PR[GP1:91,2] = PR[GP1:90,2] + -11.130;
   1:L PR[91] R[100]mm/sec CNT100;
   1:  PR[GP1:91,1] = PR[GP1:90,1] + -69.745;
   1:  PR[GP1:91,2] = PR[GP1:90,2] + -14.754;
   1:L PR[91] R[100]mm/sec CNT100;
   1:  PR[GP1:91,1] = PR[GP1:90,1] + -66.342;
   1:  PR[GP1:91,2] = PR[GP1:90,2] + -20.987;
   1:L PR[91] R[100]mm/sec CNT100;
   1:  PR[GP1:91,1] = PR[GP1:90,1] + -62.953;
   1:  PR[GP1:91,2] = PR[GP1:90,2] + -24.322;
   1:L PR[91] R[100]mm/sec CNT100;
   1:  PR[GP1:91,1] = PR[GP1:90,1] + -58.242;
   1:  PR[GP1:91,2] = PR[GP1:90,2] + -28.618;
   1:L PR[91] R[100]mm/sec CNT100;
   1:  PR[GP1:91,1] = PR[GP1:90,1] + -53.066;
   1:  PR[GP1:91,2] = PR[GP1:90,2] + -31.204;
   1:L PR[91] R[100]mm/sec CNT100;
   1:  PR[GP1:91,1] = PR[GP1:90,1] + -48.249;
   1:  PR[GP1:91,2] = PR[GP1:90,2] + -33.297;
   1:L PR[91] R[100]mm/sec CNT100;
   1:  PR[GP1:91,1] = PR[GP1:90,1] + -41.179;
   1:  PR[GP1:91,2] = PR[GP1:90,2] + -34.371;
   1:L PR[91] R[100]mm/sec CNT100;
   1:  PR[GP1:91,1] = PR[GP1:90,1] + -37.445;
   1:  PR[GP1:91,2] = PR[GP1:90,2] + -34.677;
   1:L PR[91] R[100]mm/sec CNT100;
   1:  PR[GP1:91,1] = PR[GP1:90,1] + -28.799;
   1:  PR[GP1:91,2] = PR[GP1:90,2] + -33.276;
   1:L PR[91] R[100]mm/sec CNT100;
   1:  PR[GP1:91,1] = PR[GP1:90,1] + -26.900;
   1:  PR[GP1:91,2] = PR[GP1:90,2] + -32.798;
   1:L PR[91] R[100]mm/sec CNT100;
   1:  PR[GP1:91,1] = PR[GP1:90,1] + -17.599;
   1:  PR[GP1:91,2] = PR[GP1:90,2] + -28.043;
   1:L PR[91] R[100]mm/sec CNT100;
   1:  PR[GP1:91,1] = PR[GP1:90,1] + -17.531;
   1:  PR[GP1:91,2] = PR[GP1:90,2] + -27.999;
   1:L PR[91] R[100]mm/sec CNT100;
   1:  PR[GP1:91,1] = PR[GP1:90,1] + -16.743;
   1:  PR[GP1:91,2] = PR[GP1:90,2] + -27.209;
   1:L PR[91] R[100]mm/sec CNT100;
   1:  PR[GP1:91,1] = PR[GP1:90,1] + -9.945;
   1:  PR[GP1:91,2] = PR[GP1:90,2] + -20.643;
   1:L PR[91] R[100]mm/sec CNT100;
   1:  PR[GP1:91,1] = PR[GP1:90,1] + -9.146;
   1:  PR[GP1:91,2] = PR[GP1:90,2] + -19.484;
   1:L PR[91] R[100]mm/sec CNT100;
   1:  PR[GP1:91,1] = PR[GP1:90,1] + -4.957;
   1:  PR[GP1:91,2] = PR[GP1:90,2] + -11.466;
   1:L PR[91] R[100]mm/sec CNT100;
   1:  PR[GP1:91,1] = PR[GP1:90,1] + -4.788;
   1:  PR[GP1:91,2] = PR[GP1:90,2] + -10.977;
   1:L PR[91] R[100]mm/sec CNT100;
   1:  PR[GP1:91,1] = PR[GP1:90,1] + -4.323;
   1:  PR[GP1:91,2] = PR[GP1:90,2] + -10.463;
   1:L PR[91] R[100]mm/sec CNT100;
   1:  PR[GP1:91,1] = PR[GP1:90,1] + -4.227;
   1:  PR[GP1:91,2] = PR[GP1:90,2] + -10.404;
   1:L PR[91] R[100]mm/sec CNT100;
   1:  PR[GP1:91,1] = PR[GP1:90,1] + -1.922;
   1:  PR[GP1:91,2] = PR[GP1:90,2] + -7.650;
   1:L PR[91] R[100]mm/sec CNT100;
   1:  PR[GP1:91,1] = PR[GP1:90,1] + -0.133;
   1:  PR[GP1:91,2] = PR[GP1:90,2] + -7.788;
   1:L PR[91] R[100]mm/sec CNT100;
   1:  PR[GP1:91,1] = PR[GP1:90,1] + -0.077;
   1:  PR[GP1:91,2] = PR[GP1:90,2] + -7.834;
   1:L PR[91] R[100]mm/sec CNT100;
   1:  PR[GP1:91,1] = PR[GP1:90,1] + 2.453;
   1:  PR[GP1:91,2] = PR[GP1:90,2] + -7.807;
   1:L PR[91] R[100]mm/sec CNT100;
   1:  PR[GP1:91,1] = PR[GP1:90,1] + 3.202;
   1:  PR[GP1:91,2] = PR[GP1:90,2] + -9.234;
   1:L PR[91] R[100]mm/sec CNT100;
   1:  PR[GP1:91,1] = PR[GP1:90,1] + 4.167;
   1:  PR[GP1:91,2] = PR[GP1:90,2] + -10.344;
   1:L PR[91] R[100]mm/sec CNT100;
   1:  PR[GP1:91,1] = PR[GP1:90,1] + 5.116;
   1:  PR[GP1:91,2] = PR[GP1:90,2] + -11.381;
   1:L PR[91] R[100]mm/sec CNT100;
   1:  PR[GP1:91,1] = PR[GP1:90,1] + 9.348;
   1:  PR[GP1:91,2] = PR[GP1:90,2] + -19.459;
   1:L PR[91] R[100]mm/sec CNT100;
   1:  PR[GP1:91,1] = PR[GP1:90,1] + 10.150;
   1:  PR[GP1:91,2] = PR[GP1:90,2] + -20.621;
   1:L PR[91] R[100]mm/sec CNT100;
   1:  PR[GP1:91,1] = PR[GP1:90,1] + 16.957;
   1:  PR[GP1:91,2] = PR[GP1:90,2] + -27.214;
   1:L PR[91] R[100]mm/sec CNT100;
   1:  PR[GP1:91,1] = PR[GP1:90,1] + 17.733;
   1:  PR[GP1:91,2] = PR[GP1:90,2] + -27.994;
   1:L PR[91] R[100]mm/sec CNT100;
   1:  PR[GP1:91,1] = PR[GP1:90,1] + 17.798;
   1:  PR[GP1:91,2] = PR[GP1:90,2] + -28.036;
   1:L PR[91] R[100]mm/sec CNT100;
   1:  PR[GP1:91,1] = PR[GP1:90,1] + 27.102;
   1:  PR[GP1:91,2] = PR[GP1:90,2] + -32.793;
   1:L PR[91] R[100]mm/sec CNT100;
   1:  PR[GP1:91,1] = PR[GP1:90,1] + 28.999;
   1:  PR[GP1:91,2] = PR[GP1:90,2] + -33.270;
   1:L PR[91] R[100]mm/sec CNT100;
   1:  PR[GP1:91,1] = PR[GP1:90,1] + 37.650;
   1:  PR[GP1:91,2] = PR[GP1:90,2] + -34.678;
   1:L PR[91] R[100]mm/sec CNT100;
   1:  PR[GP1:91,1] = PR[GP1:90,1] + 41.383;
   1:  PR[GP1:91,2] = PR[GP1:90,2] + -34.372;
   1:L PR[91] R[100]mm/sec CNT100;
   1:  PR[GP1:91,1] = PR[GP1:90,1] + 48.457;
   1:  PR[GP1:91,2] = PR[GP1:90,2] + -33.298;
   1:L PR[91] R[100]mm/sec CNT100;
   1:  PR[GP1:91,1] = PR[GP1:90,1] + 53.273;
   1:  PR[GP1:91,2] = PR[GP1:90,2] + -31.205;
   1:L PR[91] R[100]mm/sec CNT100;
   1:  PR[GP1:91,1] = PR[GP1:90,1] + 58.452;
   1:  PR[GP1:91,2] = PR[GP1:90,2] + -28.623;
   1:L PR[91] R[100]mm/sec CNT100;
   1:  PR[GP1:91,1] = PR[GP1:90,1] + 63.163;
   1:  PR[GP1:91,2] = PR[GP1:90,2] + -24.325;
   1:L PR[91] R[100]mm/sec CNT100;
   1:  PR[GP1:91,1] = PR[GP1:90,1] + 66.554;
   1:  PR[GP1:91,2] = PR[GP1:90,2] + -20.984;
   1:L PR[91] R[100]mm/sec CNT100;
   1:  PR[GP1:91,1] = PR[GP1:90,1] + 69.957;
   1:  PR[GP1:91,2] = PR[GP1:90,2] + -14.755;
   1:L PR[91] R[100]mm/sec CNT100;
   1:  PR[GP1:91,1] = PR[GP1:90,1] + 71.832;
   1:  PR[GP1:91,2] = PR[GP1:90,2] + -11.136;
   1:L PR[91] R[100]mm/sec CNT100;
   1:  PR[GP1:91,1] = PR[GP1:90,1] + 73.108;
   1:  PR[GP1:91,2] = PR[GP1:90,2] + -3.599;
   1:L PR[91] R[100]mm/sec CNT100;
   1:  PR[GP1:91,1] = PR[GP1:90,1] + 73.672;
   1:  PR[GP1:91,2] = PR[GP1:90,2] + -0.075;
   1:L PR[91] R[100]mm/sec CNT100;
   1:  PR[GP1:91,1] = PR[GP1:90,1] + 72.424;
   1:  PR[GP1:91,2] = PR[GP1:90,2] + 7.287;
   1:L PR[91] R[100]mm/sec CNT100;
   1:  PR[GP1:91,1] = PR[GP1:90,1] + 71.831;
   1:  PR[GP1:91,2] = PR[GP1:90,2] + 10.995;
   1:L PR[91] R[100]mm/sec CNT100;
   1:  PR[GP1:91,1] = PR[GP1:90,1] + 69.957;
   1:  PR[GP1:91,2] = PR[GP1:90,2] + 14.611;
   1:L PR[91] R[100]mm/sec CNT100;
   1:  PR[GP1:91,1] = PR[GP1:90,1] + 66.554;
   1:  PR[GP1:91,2] = PR[GP1:90,2] + 20.840;
   1:L PR[91] R[100]mm/sec CNT100;
   1:  PR[GP1:91,1] = PR[GP1:90,1] + 63.163;
   1:  PR[GP1:91,2] = PR[GP1:90,2] + 24.181;
   1:L PR[91] R[100]mm/sec CNT100;
   1:  PR[GP1:91,1] = PR[GP1:90,1] + 58.452;
   1:  PR[GP1:91,2] = PR[GP1:90,2] + 28.479;
   1:L PR[91] R[100]mm/sec CNT100;
   1:  PR[GP1:91,1] = PR[GP1:90,1] + 53.273;
   1:  PR[GP1:91,2] = PR[GP1:90,2] + 31.061;
   1:L PR[91] R[100]mm/sec CNT100;
   1:  PR[GP1:91,1] = PR[GP1:90,1] + 48.457;
   1:  PR[GP1:91,2] = PR[GP1:90,2] + 33.154;
   1:L PR[91] R[100]mm/sec CNT100;
   1:  PR[GP1:91,1] = PR[GP1:90,1] + 41.383;
   1:  PR[GP1:91,2] = PR[GP1:90,2] + 34.228;
   1:L PR[91] R[100]mm/sec CNT100;
   1:  PR[GP1:91,1] = PR[GP1:90,1] + 37.650;
   1:  PR[GP1:91,2] = PR[GP1:90,2] + 34.534;
   1:L PR[91] R[100]mm/sec CNT100;
   1:  PR[GP1:91,1] = PR[GP1:90,1] + 28.999;
   1:  PR[GP1:91,2] = PR[GP1:90,2] + 33.126;
   1:L PR[91] R[100]mm/sec CNT100;
   1:  PR[GP1:91,1] = PR[GP1:90,1] + 27.102;
   1:  PR[GP1:91,2] = PR[GP1:90,2] + 32.649;
   1:L PR[91] R[100]mm/sec CNT100;
   1:  PR[GP1:91,1] = PR[GP1:90,1] + 17.798;
   1:  PR[GP1:91,2] = PR[GP1:90,2] + 27.892;
   1:L PR[91] R[100]mm/sec CNT100;
   1:  PR[GP1:91,1] = PR[GP1:90,1] + 17.733;
   1:  PR[GP1:91,2] = PR[GP1:90,2] + 27.849;
   1:L PR[91] R[100]mm/sec CNT100;
   1:  PR[GP1:91,1] = PR[GP1:90,1] + 16.957;
   1:  PR[GP1:91,2] = PR[GP1:90,2] + 27.070;
   1:L PR[91] R[100]mm/sec CNT100;
   1:  PR[GP1:91,1] = PR[GP1:90,1] + 10.149;
   1:  PR[GP1:91,2] = PR[GP1:90,2] + 20.477;
   1:L PR[91] R[100]mm/sec CNT100;
   1:  PR[GP1:91,1] = PR[GP1:90,1] + 9.351;
   1:  PR[GP1:91,2] = PR[GP1:90,2] + 19.321;
   1:L PR[91] R[100]mm/sec CNT100;
   1:  PR[GP1:91,1] = PR[GP1:90,1] + 5.173;
   1:  PR[GP1:91,2] = PR[GP1:90,2] + 11.346;
   1:L PR[91] R[100]mm/sec CNT100;
   1:  PR[GP1:91,1] = PR[GP1:90,1] + 4.992;
   1:  PR[GP1:91,2] = PR[GP1:90,2] + 10.820;
   1:L PR[91] R[100]mm/sec CNT100;
   1:  PR[GP1:91,1] = PR[GP1:90,1] + 2.976;
   1:  PR[GP1:91,2] = PR[GP1:90,2] + 8.378;
   1:L PR[91] R[100]mm/sec CNT100;
   1:  PR[GP1:91,1] = PR[GP1:90,1] + 2.376;
   1:  PR[GP1:91,2] = PR[GP1:90,2] + 7.725;
   1:L PR[91] R[100]mm/sec CNT100;
   1:  PR[GP1:91,1] = PR[GP1:90,1] + 1.972;
   1:  PR[GP1:91,2] = PR[GP1:90,2] + 7.502;
   1:L PR[91] R[100]mm/sec CNT100;
   1:  PR[GP1:91,1] = PR[GP1:90,1] + -0.552;
   1:  PR[GP1:91,2] = PR[GP1:90,2] + 7.528;
   1:L PR[91] R[100]mm/sec CNT100;
   1:  ! -- Layer/Ebene 40 -- !;
   1:  PR[91] = PR[90];
   1:  PR[GP1:91,1] = PR[GP1:90,1] + -2.026;
   1:  PR[GP1:91,2] = PR[GP1:90,2] + 8.156;
   1:  PR[GP1:91,3] = PR[GP1:90,3] + 24.705;
   1:L PR[91] R[100]mm/sec CNT100;
   1:  PR[GP1:91,1] = PR[GP1:90,1] + -2.304;
   1:  PR[GP1:91,2] = PR[GP1:90,2] + 8.351;
   1:L PR[91] R[100]mm/sec CNT100;
   1:  PR[GP1:91,1] = PR[GP1:90,1] + -4.616;
   1:  PR[GP1:91,2] = PR[GP1:90,2] + 11.184;
   1:L PR[91] R[100]mm/sec CNT100;
   1:  PR[GP1:91,1] = PR[GP1:90,1] + -4.912;
   1:  PR[GP1:91,2] = PR[GP1:90,2] + 11.717;
   1:L PR[91] R[100]mm/sec CNT100;
   1:  PR[GP1:91,1] = PR[GP1:90,1] + -8.638;
   1:  PR[GP1:91,2] = PR[GP1:90,2] + 18.834;
   1:L PR[91] R[100]mm/sec CNT100;
   1:  PR[GP1:91,1] = PR[GP1:90,1] + -9.989;
   1:  PR[GP1:91,2] = PR[GP1:90,2] + 20.791;
   1:L PR[91] R[100]mm/sec CNT100;
   1:  PR[GP1:91,1] = PR[GP1:90,1] + -17.039;
   1:  PR[GP1:91,2] = PR[GP1:90,2] + 27.600;
   1:L PR[91] R[100]mm/sec CNT100;
   1:  PR[GP1:91,1] = PR[GP1:90,1] + -17.553;
   1:  PR[GP1:91,2] = PR[GP1:90,2] + 27.997;
   1:L PR[91] R[100]mm/sec CNT100;
   1:  PR[GP1:91,1] = PR[GP1:90,1] + -21.092;
   1:  PR[GP1:91,2] = PR[GP1:90,2] + 29.723;
   1:L PR[91] R[100]mm/sec CNT100;
   1:  PR[GP1:91,1] = PR[GP1:90,1] + -27.029;
   1:  PR[GP1:91,2] = PR[GP1:90,2] + 32.758;
   1:L PR[91] R[100]mm/sec CNT100;
   1:  PR[GP1:91,1] = PR[GP1:90,1] + -28.088;
   1:  PR[GP1:91,2] = PR[GP1:90,2] + 33.025;
   1:L PR[91] R[100]mm/sec CNT100;
   1:  PR[GP1:91,1] = PR[GP1:90,1] + -37.544;
   1:  PR[GP1:91,2] = PR[GP1:90,2] + 34.558;
   1:L PR[91] R[100]mm/sec CNT100;
   1:  PR[GP1:91,1] = PR[GP1:90,1] + -40.481;
   1:  PR[GP1:91,2] = PR[GP1:90,2] + 34.317;
   1:L PR[91] R[100]mm/sec CNT100;
   1:  PR[GP1:91,1] = PR[GP1:90,1] + -48.304;
   1:  PR[GP1:91,2] = PR[GP1:90,2] + 33.129;
   1:L PR[91] R[100]mm/sec CNT100;
   1:  PR[GP1:91,1] = PR[GP1:90,1] + -52.442;
   1:  PR[GP1:91,2] = PR[GP1:90,2] + 31.330;
   1:L PR[91] R[100]mm/sec CNT100;
   1:  PR[GP1:91,1] = PR[GP1:90,1] + -58.251;
   1:  PR[GP1:91,2] = PR[GP1:90,2] + 28.429;
   1:L PR[91] R[100]mm/sec CNT100;
   1:  PR[GP1:91,1] = PR[GP1:90,1] + -62.454;
   1:  PR[GP1:91,2] = PR[GP1:90,2] + 24.596;
   1:L PR[91] R[100]mm/sec CNT100;
   1:  PR[GP1:91,1] = PR[GP1:90,1] + -66.311;
   1:  PR[GP1:91,2] = PR[GP1:90,2] + 20.800;
   1:L PR[91] R[100]mm/sec CNT100;
   1:  PR[GP1:91,1] = PR[GP1:90,1] + -69.405;
   1:  PR[GP1:91,2] = PR[GP1:90,2] + 15.133;
   1:L PR[91] R[100]mm/sec CNT100;
   1:  PR[GP1:91,1] = PR[GP1:90,1] + -71.563;
   1:  PR[GP1:91,2] = PR[GP1:90,2] + 10.958;
   1:L PR[91] R[100]mm/sec CNT100;
   1:  PR[GP1:91,1] = PR[GP1:90,1] + -72.733;
   1:  PR[GP1:91,2] = PR[GP1:90,2] + 4.046;
   1:L PR[91] R[100]mm/sec CNT100;
   1:  PR[GP1:91,1] = PR[GP1:90,1] + -73.392;
   1:  PR[GP1:91,2] = PR[GP1:90,2] + -0.069;
   1:L PR[91] R[100]mm/sec CNT100;
   1:  PR[GP1:91,1] = PR[GP1:90,1] + -72.243;
   1:  PR[GP1:91,2] = PR[GP1:90,2] + -6.843;
   1:L PR[91] R[100]mm/sec CNT100;
   1:  PR[GP1:91,1] = PR[GP1:90,1] + -71.561;
   1:  PR[GP1:91,2] = PR[GP1:90,2] + -11.104;
   1:L PR[91] R[100]mm/sec CNT100;
   1:  PR[GP1:91,1] = PR[GP1:90,1] + -69.405;
   1:  PR[GP1:91,2] = PR[GP1:90,2] + -15.277;
   1:L PR[91] R[100]mm/sec CNT100;
   1:  PR[GP1:91,1] = PR[GP1:90,1] + -66.311;
   1:  PR[GP1:91,2] = PR[GP1:90,2] + -20.944;
   1:L PR[91] R[100]mm/sec CNT100;
   1:  PR[GP1:91,1] = PR[GP1:90,1] + -62.454;
   1:  PR[GP1:91,2] = PR[GP1:90,2] + -24.740;
   1:L PR[91] R[100]mm/sec CNT100;
   1:  PR[GP1:91,1] = PR[GP1:90,1] + -58.251;
   1:  PR[GP1:91,2] = PR[GP1:90,2] + -28.573;
   1:L PR[91] R[100]mm/sec CNT100;
   1:  PR[GP1:91,1] = PR[GP1:90,1] + -52.442;
   1:  PR[GP1:91,2] = PR[GP1:90,2] + -31.474;
   1:L PR[91] R[100]mm/sec CNT100;
   1:  PR[GP1:91,1] = PR[GP1:90,1] + -48.304;
   1:  PR[GP1:91,2] = PR[GP1:90,2] + -33.273;
   1:L PR[91] R[100]mm/sec CNT100;
   1:  PR[GP1:91,1] = PR[GP1:90,1] + -40.481;
   1:  PR[GP1:91,2] = PR[GP1:90,2] + -34.461;
   1:L PR[91] R[100]mm/sec CNT100;
   1:  PR[GP1:91,1] = PR[GP1:90,1] + -37.544;
   1:  PR[GP1:91,2] = PR[GP1:90,2] + -34.702;
   1:L PR[91] R[100]mm/sec CNT100;
   1:  PR[GP1:91,1] = PR[GP1:90,1] + -28.088;
   1:  PR[GP1:91,2] = PR[GP1:90,2] + -33.169;
   1:L PR[91] R[100]mm/sec CNT100;
   1:  PR[GP1:91,1] = PR[GP1:90,1] + -27.029;
   1:  PR[GP1:91,2] = PR[GP1:90,2] + -32.902;
   1:L PR[91] R[100]mm/sec CNT100;
   1:  PR[GP1:91,1] = PR[GP1:90,1] + -21.092;
   1:  PR[GP1:91,2] = PR[GP1:90,2] + -29.867;
   1:L PR[91] R[100]mm/sec CNT100;
   1:  PR[GP1:91,1] = PR[GP1:90,1] + -17.553;
   1:  PR[GP1:91,2] = PR[GP1:90,2] + -28.141;
   1:L PR[91] R[100]mm/sec CNT100;
   1:  PR[GP1:91,1] = PR[GP1:90,1] + -17.039;
   1:  PR[GP1:91,2] = PR[GP1:90,2] + -27.744;
   1:L PR[91] R[100]mm/sec CNT100;
   1:  PR[GP1:91,1] = PR[GP1:90,1] + -9.989;
   1:  PR[GP1:91,2] = PR[GP1:90,2] + -20.935;
   1:L PR[91] R[100]mm/sec CNT100;
   1:  PR[GP1:91,1] = PR[GP1:90,1] + -8.632;
   1:  PR[GP1:91,2] = PR[GP1:90,2] + -18.968;
   1:L PR[91] R[100]mm/sec CNT100;
   1:  PR[GP1:91,1] = PR[GP1:90,1] + -4.921;
   1:  PR[GP1:91,2] = PR[GP1:90,2] + -11.864;
   1:L PR[91] R[100]mm/sec CNT100;
   1:  PR[GP1:91,1] = PR[GP1:90,1] + -4.822;
   1:  PR[GP1:91,2] = PR[GP1:90,2] + -11.577;
   1:L PR[91] R[100]mm/sec CNT100;
   1:  PR[GP1:91,1] = PR[GP1:90,1] + -4.702;
   1:  PR[GP1:91,2] = PR[GP1:90,2] + -11.445;
   1:L PR[91] R[100]mm/sec CNT100;
   1:  PR[GP1:91,1] = PR[GP1:90,1] + -4.676;
   1:  PR[GP1:91,2] = PR[GP1:90,2] + -11.395;
   1:L PR[91] R[100]mm/sec CNT100;
   1:  PR[GP1:91,1] = PR[GP1:90,1] + -4.661;
   1:  PR[GP1:91,2] = PR[GP1:90,2] + -11.400;
   1:L PR[91] R[100]mm/sec CNT100;
   1:  PR[GP1:91,1] = PR[GP1:90,1] + -4.494;
   1:  PR[GP1:91,2] = PR[GP1:90,2] + -11.215;
   1:L PR[91] R[100]mm/sec CNT100;
   1:  PR[GP1:91,1] = PR[GP1:90,1] + -4.443;
   1:  PR[GP1:91,2] = PR[GP1:90,2] + -11.183;
   1:L PR[91] R[100]mm/sec CNT100;
   1:  PR[GP1:91,1] = PR[GP1:90,1] + -1.932;
   1:  PR[GP1:91,2] = PR[GP1:90,2] + -8.183;
   1:L PR[91] R[100]mm/sec CNT100;
   1:  PR[GP1:91,1] = PR[GP1:90,1] + -0.380;
   1:  PR[GP1:91,2] = PR[GP1:90,2] + -8.302;
   1:L PR[91] R[100]mm/sec CNT100;
   1:  PR[GP1:91,1] = PR[GP1:90,1] + -0.338;
   1:  PR[GP1:91,2] = PR[GP1:90,2] + -8.337;
   1:L PR[91] R[100]mm/sec CNT100;
   1:  PR[GP1:91,1] = PR[GP1:90,1] + 2.408;
   1:  PR[GP1:91,2] = PR[GP1:90,2] + -8.308;
   1:L PR[91] R[100]mm/sec CNT100;
   1:  PR[GP1:91,1] = PR[GP1:90,1] + 3.046;
   1:  PR[GP1:91,2] = PR[GP1:90,2] + -9.523;
   1:L PR[91] R[100]mm/sec CNT100;
   1:  PR[GP1:91,1] = PR[GP1:90,1] + 3.825;
   1:  PR[GP1:91,2] = PR[GP1:90,2] + -10.420;
   1:L PR[91] R[100]mm/sec CNT100;
   1:  PR[GP1:91,1] = PR[GP1:90,1] + 5.085;
   1:  PR[GP1:91,2] = PR[GP1:90,2] + -11.793;
   1:L PR[91] R[100]mm/sec CNT100;
   1:  PR[GP1:91,1] = PR[GP1:90,1] + 8.835;
   1:  PR[GP1:91,2] = PR[GP1:90,2] + -18.944;
   1:L PR[91] R[100]mm/sec CNT100;
   1:  PR[GP1:91,1] = PR[GP1:90,1] + 10.194;
   1:  PR[GP1:91,2] = PR[GP1:90,2] + -20.915;
   1:L PR[91] R[100]mm/sec CNT100;
   1:  PR[GP1:91,1] = PR[GP1:90,1] + 17.239;
   1:  PR[GP1:91,2] = PR[GP1:90,2] + -27.738;
   1:L PR[91] R[100]mm/sec CNT100;
   1:  PR[GP1:91,1] = PR[GP1:90,1] + 17.755;
   1:  PR[GP1:91,2] = PR[GP1:90,2] + -28.136;
   1:L PR[91] R[100]mm/sec CNT100;
   1:  PR[GP1:91,1] = PR[GP1:90,1] + 21.305;
   1:  PR[GP1:91,2] = PR[GP1:90,2] + -29.867;
   1:L PR[91] R[100]mm/sec CNT100;
   1:  PR[GP1:91,1] = PR[GP1:90,1] + 27.230;
   1:  PR[GP1:91,2] = PR[GP1:90,2] + -32.897;
   1:L PR[91] R[100]mm/sec CNT100;
   1:  PR[GP1:91,1] = PR[GP1:90,1] + 28.288;
   1:  PR[GP1:91,2] = PR[GP1:90,2] + -33.163;
   1:L PR[91] R[100]mm/sec CNT100;
   1:  PR[GP1:91,1] = PR[GP1:90,1] + 37.749;
   1:  PR[GP1:91,2] = PR[GP1:90,2] + -34.702;
   1:L PR[91] R[100]mm/sec CNT100;
   1:  PR[GP1:91,1] = PR[GP1:90,1] + 40.684;
   1:  PR[GP1:91,2] = PR[GP1:90,2] + -34.461;
   1:L PR[91] R[100]mm/sec CNT100;
   1:  PR[GP1:91,1] = PR[GP1:90,1] + 48.511;
   1:  PR[GP1:91,2] = PR[GP1:90,2] + -33.273;
   1:L PR[91] R[100]mm/sec CNT100;
   1:  PR[GP1:91,1] = PR[GP1:90,1] + 52.649;
   1:  PR[GP1:91,2] = PR[GP1:90,2] + -31.475;
   1:L PR[91] R[100]mm/sec CNT100;
   1:  PR[GP1:91,1] = PR[GP1:90,1] + 58.460;
   1:  PR[GP1:91,2] = PR[GP1:90,2] + -28.578;
   1:L PR[91] R[100]mm/sec CNT100;
   1:  PR[GP1:91,1] = PR[GP1:90,1] + 62.663;
   1:  PR[GP1:91,2] = PR[GP1:90,2] + -24.743;
   1:L PR[91] R[100]mm/sec CNT100;
   1:  PR[GP1:91,1] = PR[GP1:90,1] + 66.522;
   1:  PR[GP1:91,2] = PR[GP1:90,2] + -20.940;
   1:L PR[91] R[100]mm/sec CNT100;
   1:  PR[GP1:91,1] = PR[GP1:90,1] + 69.617;
   1:  PR[GP1:91,2] = PR[GP1:90,2] + -15.277;
   1:L PR[91] R[100]mm/sec CNT100;
   1:  PR[GP1:91,1] = PR[GP1:90,1] + 71.776;
   1:  PR[GP1:91,2] = PR[GP1:90,2] + -11.112;
   1:L PR[91] R[100]mm/sec CNT100;
   1:  PR[GP1:91,1] = PR[GP1:90,1] + 72.946;
   1:  PR[GP1:91,2] = PR[GP1:90,2] + -4.197;
   1:L PR[91] R[100]mm/sec CNT100;
   1:  PR[GP1:91,1] = PR[GP1:90,1] + 73.605;
   1:  PR[GP1:91,2] = PR[GP1:90,2] + -0.075;
   1:L PR[91] R[100]mm/sec CNT100;
   1:  PR[GP1:91,1] = PR[GP1:90,1] + 72.456;
   1:  PR[GP1:91,2] = PR[GP1:90,2] + 6.702;
   1:L PR[91] R[100]mm/sec CNT100;
   1:  PR[GP1:91,1] = PR[GP1:90,1] + 71.774;
   1:  PR[GP1:91,2] = PR[GP1:90,2] + 10.970;
   1:L PR[91] R[100]mm/sec CNT100;
   1:  PR[GP1:91,1] = PR[GP1:90,1] + 69.617;
   1:  PR[GP1:91,2] = PR[GP1:90,2] + 15.133;
   1:L PR[91] R[100]mm/sec CNT100;
   1:  PR[GP1:91,1] = PR[GP1:90,1] + 66.522;
   1:  PR[GP1:91,2] = PR[GP1:90,2] + 20.796;
   1:L PR[91] R[100]mm/sec CNT100;
   1:  PR[GP1:91,1] = PR[GP1:90,1] + 62.663;
   1:  PR[GP1:91,2] = PR[GP1:90,2] + 24.599;
   1:L PR[91] R[100]mm/sec CNT100;
   1:  PR[GP1:91,1] = PR[GP1:90,1] + 58.460;
   1:  PR[GP1:91,2] = PR[GP1:90,2] + 28.434;
   1:L PR[91] R[100]mm/sec CNT100;
   1:  PR[GP1:91,1] = PR[GP1:90,1] + 52.649;
   1:  PR[GP1:91,2] = PR[GP1:90,2] + 31.331;
   1:L PR[91] R[100]mm/sec CNT100;
   1:  PR[GP1:91,1] = PR[GP1:90,1] + 48.511;
   1:  PR[GP1:91,2] = PR[GP1:90,2] + 33.129;
   1:L PR[91] R[100]mm/sec CNT100;
   1:  PR[GP1:91,1] = PR[GP1:90,1] + 40.684;
   1:  PR[GP1:91,2] = PR[GP1:90,2] + 34.317;
   1:L PR[91] R[100]mm/sec CNT100;
   1:  PR[GP1:91,1] = PR[GP1:90,1] + 37.749;
   1:  PR[GP1:91,2] = PR[GP1:90,2] + 34.558;
   1:L PR[91] R[100]mm/sec CNT100;
   1:  PR[GP1:91,1] = PR[GP1:90,1] + 28.288;
   1:  PR[GP1:91,2] = PR[GP1:90,2] + 33.019;
   1:L PR[91] R[100]mm/sec CNT100;
   1:  PR[GP1:91,1] = PR[GP1:90,1] + 27.230;
   1:  PR[GP1:91,2] = PR[GP1:90,2] + 32.753;
   1:L PR[91] R[100]mm/sec CNT100;
   1:  PR[GP1:91,1] = PR[GP1:90,1] + 21.305;
   1:  PR[GP1:91,2] = PR[GP1:90,2] + 29.723;
   1:L PR[91] R[100]mm/sec CNT100;
   1:  PR[GP1:91,1] = PR[GP1:90,1] + 17.754;
   1:  PR[GP1:91,2] = PR[GP1:90,2] + 27.992;
   1:L PR[91] R[100]mm/sec CNT100;
   1:  PR[GP1:91,1] = PR[GP1:90,1] + 17.239;
   1:  PR[GP1:91,2] = PR[GP1:90,2] + 27.594;
   1:L PR[91] R[100]mm/sec CNT100;
   1:  PR[GP1:91,1] = PR[GP1:90,1] + 10.194;
   1:  PR[GP1:91,2] = PR[GP1:90,2] + 20.771;
   1:L PR[91] R[100]mm/sec CNT100;
   1:  PR[GP1:91,1] = PR[GP1:90,1] + 8.840;
   1:  PR[GP1:91,2] = PR[GP1:90,2] + 18.810;
   1:L PR[91] R[100]mm/sec CNT100;
   1:  PR[GP1:91,1] = PR[GP1:90,1] + 5.142;
   1:  PR[GP1:91,2] = PR[GP1:90,2] + 11.758;
   1:L PR[91] R[100]mm/sec CNT100;
   1:  PR[GP1:91,1] = PR[GP1:90,1] + 5.025;
   1:  PR[GP1:91,2] = PR[GP1:90,2] + 11.418;
   1:L PR[91] R[100]mm/sec CNT100;
   1:  PR[GP1:91,1] = PR[GP1:90,1] + 2.853;
   1:  PR[GP1:91,2] = PR[GP1:90,2] + 8.786;
   1:L PR[91] R[100]mm/sec CNT100;
   1:  PR[GP1:91,1] = PR[GP1:90,1] + 2.348;
   1:  PR[GP1:91,2] = PR[GP1:90,2] + 8.238;
   1:L PR[91] R[100]mm/sec CNT100;
   1:  PR[GP1:91,1] = PR[GP1:90,1] + 1.977;
   1:  PR[GP1:91,2] = PR[GP1:90,2] + 8.032;
   1:L PR[91] R[100]mm/sec CNT100;
   1:  PR[GP1:91,1] = PR[GP1:90,1] + -0.770;
   1:  PR[GP1:91,2] = PR[GP1:90,2] + 8.061;
   1:L PR[91] R[100]mm/sec CNT100;
   1:  ! -- Layer/Ebene 41 -- !;
   1:  PR[91] = PR[90];
   1:  PR[GP1:91,1] = PR[GP1:90,1] + -2.003;
   1:  PR[GP1:91,2] = PR[GP1:90,2] + 8.671;
   1:  PR[GP1:91,3] = PR[GP1:90,3] + 25.315;
   1:L PR[91] R[100]mm/sec CNT100;
   1:  PR[GP1:91,1] = PR[GP1:90,1] + -2.264;
   1:  PR[GP1:91,2] = PR[GP1:90,2] + 8.854;
   1:L PR[91] R[100]mm/sec CNT100;
   1:  PR[GP1:91,1] = PR[GP1:90,1] + -4.766;
   1:  PR[GP1:91,2] = PR[GP1:90,2] + 11.920;
   1:L PR[91] R[100]mm/sec CNT100;
   1:  PR[GP1:91,1] = PR[GP1:90,1] + -8.126;
   1:  PR[GP1:91,2] = PR[GP1:90,2] + 18.322;
   1:L PR[91] R[100]mm/sec CNT100;
   1:  PR[GP1:91,1] = PR[GP1:90,1] + -10.033;
   1:  PR[GP1:91,2] = PR[GP1:90,2] + 21.083;
   1:L PR[91] R[100]mm/sec CNT100;
   1:  PR[GP1:91,1] = PR[GP1:90,1] + -16.387;
   1:  PR[GP1:91,2] = PR[GP1:90,2] + 27.220;
   1:L PR[91] R[100]mm/sec CNT100;
   1:  PR[GP1:91,1] = PR[GP1:90,1] + -17.626;
   1:  PR[GP1:91,2] = PR[GP1:90,2] + 28.177;
   1:L PR[91] R[100]mm/sec CNT100;
   1:  PR[GP1:91,1] = PR[GP1:90,1] + -25.592;
   1:  PR[GP1:91,2] = PR[GP1:90,2] + 32.062;
   1:L PR[91] R[100]mm/sec CNT100;
   1:  PR[GP1:91,1] = PR[GP1:90,1] + -27.158;
   1:  PR[GP1:91,2] = PR[GP1:90,2] + 32.863;
   1:L PR[91] R[100]mm/sec CNT100;
   1:  PR[GP1:91,1] = PR[GP1:90,1] + -27.378;
   1:  PR[GP1:91,2] = PR[GP1:90,2] + 32.918;
   1:L PR[91] R[100]mm/sec CNT100;
   1:  PR[GP1:91,1] = PR[GP1:90,1] + -37.644;
   1:  PR[GP1:91,2] = PR[GP1:90,2] + 34.582;
   1:L PR[91] R[100]mm/sec CNT100;
   1:  PR[GP1:91,1] = PR[GP1:90,1] + -39.782;
   1:  PR[GP1:91,2] = PR[GP1:90,2] + 34.407;
   1:L PR[91] R[100]mm/sec CNT100;
   1:  PR[GP1:91,1] = PR[GP1:90,1] + -48.359;
   1:  PR[GP1:91,2] = PR[GP1:90,2] + 33.104;
   1:L PR[91] R[100]mm/sec CNT100;
   1:  PR[GP1:91,1] = PR[GP1:90,1] + -51.819;
   1:  PR[GP1:91,2] = PR[GP1:90,2] + 31.600;
   1:L PR[91] R[100]mm/sec CNT100;
   1:  PR[GP1:91,1] = PR[GP1:90,1] + -58.259;
   1:  PR[GP1:91,2] = PR[GP1:90,2] + 28.384;
   1:L PR[91] R[100]mm/sec CNT100;
   1:  PR[GP1:91,1] = PR[GP1:90,1] + -61.954;
   1:  PR[GP1:91,2] = PR[GP1:90,2] + 25.013;
   1:L PR[91] R[100]mm/sec CNT100;
   1:  PR[GP1:91,1] = PR[GP1:90,1] + -66.280;
   1:  PR[GP1:91,2] = PR[GP1:90,2] + 20.756;
   1:L PR[91] R[100]mm/sec CNT100;
   1:  PR[GP1:91,1] = PR[GP1:90,1] + -69.065;
   1:  PR[GP1:91,2] = PR[GP1:90,2] + 15.656;
   1:L PR[91] R[100]mm/sec CNT100;
   1:  PR[GP1:91,1] = PR[GP1:90,1] + -71.506;
   1:  PR[GP1:91,2] = PR[GP1:90,2] + 10.932;
   1:L PR[91] R[100]mm/sec CNT100;
   1:  PR[GP1:91,1] = PR[GP1:90,1] + -72.571;
   1:  PR[GP1:91,2] = PR[GP1:90,2] + 4.642;
   1:L PR[91] R[100]mm/sec CNT100;
   1:  PR[GP1:91,1] = PR[GP1:90,1] + -73.326;
   1:  PR[GP1:91,2] = PR[GP1:90,2] + -0.069;
   1:L PR[91] R[100]mm/sec CNT100;
   1:  PR[GP1:91,1] = PR[GP1:90,1] + -72.276;
   1:  PR[GP1:91,2] = PR[GP1:90,2] + -6.258;
   1:L PR[91] R[100]mm/sec CNT100;
   1:  PR[GP1:91,1] = PR[GP1:90,1] + -71.505;
   1:  PR[GP1:91,2] = PR[GP1:90,2] + -11.079;
   1:L PR[91] R[100]mm/sec CNT100;
   1:  PR[GP1:91,1] = PR[GP1:90,1] + -69.065;
   1:  PR[GP1:91,2] = PR[GP1:90,2] + -15.800;
   1:L PR[91] R[100]mm/sec CNT100;
   1:  PR[GP1:91,1] = PR[GP1:90,1] + -66.280;
   1:  PR[GP1:91,2] = PR[GP1:90,2] + -20.900;
   1:L PR[91] R[100]mm/sec CNT100;
   1:  PR[GP1:91,1] = PR[GP1:90,1] + -61.954;
   1:  PR[GP1:91,2] = PR[GP1:90,2] + -25.157;
   1:L PR[91] R[100]mm/sec CNT100;
   1:  PR[GP1:91,1] = PR[GP1:90,1] + -58.259;
   1:  PR[GP1:91,2] = PR[GP1:90,2] + -28.528;
   1:L PR[91] R[100]mm/sec CNT100;
   1:  PR[GP1:91,1] = PR[GP1:90,1] + -51.819;
   1:  PR[GP1:91,2] = PR[GP1:90,2] + -31.744;
   1:L PR[91] R[100]mm/sec CNT100;
   1:  PR[GP1:91,1] = PR[GP1:90,1] + -48.359;
   1:  PR[GP1:91,2] = PR[GP1:90,2] + -33.248;
   1:L PR[91] R[100]mm/sec CNT100;
   1:  PR[GP1:91,1] = PR[GP1:90,1] + -39.782;
   1:  PR[GP1:91,2] = PR[GP1:90,2] + -34.551;
   1:L PR[91] R[100]mm/sec CNT100;
   1:  PR[GP1:91,1] = PR[GP1:90,1] + -37.644;
   1:  PR[GP1:91,2] = PR[GP1:90,2] + -34.726;
   1:L PR[91] R[100]mm/sec CNT100;
   1:  PR[GP1:91,1] = PR[GP1:90,1] + -27.378;
   1:  PR[GP1:91,2] = PR[GP1:90,2] + -33.062;
   1:L PR[91] R[100]mm/sec CNT100;
   1:  PR[GP1:91,1] = PR[GP1:90,1] + -27.158;
   1:  PR[GP1:91,2] = PR[GP1:90,2] + -33.007;
   1:L PR[91] R[100]mm/sec CNT100;
   1:  PR[GP1:91,1] = PR[GP1:90,1] + -25.592;
   1:  PR[GP1:91,2] = PR[GP1:90,2] + -32.206;
   1:L PR[91] R[100]mm/sec CNT100;
   1:  PR[GP1:91,1] = PR[GP1:90,1] + -17.626;
   1:  PR[GP1:91,2] = PR[GP1:90,2] + -28.321;
   1:L PR[91] R[100]mm/sec CNT100;
   1:  PR[GP1:91,1] = PR[GP1:90,1] + -16.387;
   1:  PR[GP1:91,2] = PR[GP1:90,2] + -27.364;
   1:L PR[91] R[100]mm/sec CNT100;
   1:  PR[GP1:91,1] = PR[GP1:90,1] + -10.033;
   1:  PR[GP1:91,2] = PR[GP1:90,2] + -21.227;
   1:L PR[91] R[100]mm/sec CNT100;
   1:  PR[GP1:91,1] = PR[GP1:90,1] + -8.119;
   1:  PR[GP1:91,2] = PR[GP1:90,2] + -18.452;
   1:L PR[91] R[100]mm/sec CNT100;
   1:  PR[GP1:91,1] = PR[GP1:90,1] + -4.885;
   1:  PR[GP1:91,2] = PR[GP1:90,2] + -12.261;
   1:L PR[91] R[100]mm/sec CNT100;
   1:  PR[GP1:91,1] = PR[GP1:90,1] + -4.860;
   1:  PR[GP1:91,2] = PR[GP1:90,2] + -12.188;
   1:L PR[91] R[100]mm/sec CNT100;
   1:  PR[GP1:91,1] = PR[GP1:90,1] + -4.826;
   1:  PR[GP1:91,2] = PR[GP1:90,2] + -12.148;
   1:L PR[91] R[100]mm/sec CNT100;
   1:  PR[GP1:91,1] = PR[GP1:90,1] + -4.644;
   1:  PR[GP1:91,2] = PR[GP1:90,2] + -11.800;
   1:L PR[91] R[100]mm/sec CNT100;
   1:  PR[GP1:91,1] = PR[GP1:90,1] + -4.558;
   1:  PR[GP1:91,2] = PR[GP1:90,2] + -11.829;
   1:L PR[91] R[100]mm/sec CNT100;
   1:  PR[GP1:91,1] = PR[GP1:90,1] + -1.941;
   1:  PR[GP1:91,2] = PR[GP1:90,2] + -8.716;
   1:L PR[91] R[100]mm/sec CNT100;
   1:  PR[GP1:91,1] = PR[GP1:90,1] + -0.627;
   1:  PR[GP1:91,2] = PR[GP1:90,2] + -8.817;
   1:L PR[91] R[100]mm/sec CNT100;
   1:  PR[GP1:91,1] = PR[GP1:90,1] + -0.600;
   1:  PR[GP1:91,2] = PR[GP1:90,2] + -8.840;
   1:L PR[91] R[100]mm/sec CNT100;
   1:  PR[GP1:91,1] = PR[GP1:90,1] + 2.363;
   1:  PR[GP1:91,2] = PR[GP1:90,2] + -8.809;
   1:L PR[91] R[100]mm/sec CNT100;
   1:  PR[GP1:91,1] = PR[GP1:90,1] + 2.890;
   1:  PR[GP1:91,2] = PR[GP1:90,2] + -9.811;
   1:L PR[91] R[100]mm/sec CNT100;
   1:  PR[GP1:91,1] = PR[GP1:90,1] + 3.484;
   1:  PR[GP1:91,2] = PR[GP1:90,2] + -10.495;
   1:L PR[91] R[100]mm/sec CNT100;
   1:  PR[GP1:91,1] = PR[GP1:90,1] + 5.053;
   1:  PR[GP1:91,2] = PR[GP1:90,2] + -12.205;
   1:L PR[91] R[100]mm/sec CNT100;
   1:  PR[GP1:91,1] = PR[GP1:90,1] + 8.322;
   1:  PR[GP1:91,2] = PR[GP1:90,2] + -18.429;
   1:L PR[91] R[100]mm/sec CNT100;
   1:  PR[GP1:91,1] = PR[GP1:90,1] + 10.239;
   1:  PR[GP1:91,2] = PR[GP1:90,2] + -21.209;
   1:L PR[91] R[100]mm/sec CNT100;
   1:  PR[GP1:91,1] = PR[GP1:90,1] + 16.588;
   1:  PR[GP1:91,2] = PR[GP1:90,2] + -27.357;
   1:L PR[91] R[100]mm/sec CNT100;
   1:  PR[GP1:91,1] = PR[GP1:90,1] + 17.829;
   1:  PR[GP1:91,2] = PR[GP1:90,2] + -28.316;
   1:L PR[91] R[100]mm/sec CNT100;
   1:  PR[GP1:91,1] = PR[GP1:90,1] + 25.805;
   1:  PR[GP1:91,2] = PR[GP1:90,2] + -32.206;
   1:L PR[91] R[100]mm/sec CNT100;
   1:  PR[GP1:91,1] = PR[GP1:90,1] + 27.359;
   1:  PR[GP1:91,2] = PR[GP1:90,2] + -33.001;
   1:L PR[91] R[100]mm/sec CNT100;
   1:  PR[GP1:91,1] = PR[GP1:90,1] + 27.577;
   1:  PR[GP1:91,2] = PR[GP1:90,2] + -33.056;
   1:L PR[91] R[100]mm/sec CNT100;
   1:  PR[GP1:91,1] = PR[GP1:90,1] + 37.848;
   1:  PR[GP1:91,2] = PR[GP1:90,2] + -34.726;
   1:L PR[91] R[100]mm/sec CNT100;
   1:  PR[GP1:91,1] = PR[GP1:90,1] + 39.985;
   1:  PR[GP1:91,2] = PR[GP1:90,2] + -34.551;
   1:L PR[91] R[100]mm/sec CNT100;
   1:  PR[GP1:91,1] = PR[GP1:90,1] + 48.566;
   1:  PR[GP1:91,2] = PR[GP1:90,2] + -33.249;
   1:L PR[91] R[100]mm/sec CNT100;
   1:  PR[GP1:91,1] = PR[GP1:90,1] + 52.025;
   1:  PR[GP1:91,2] = PR[GP1:90,2] + -31.745;
   1:L PR[91] R[100]mm/sec CNT100;
   1:  PR[GP1:91,1] = PR[GP1:90,1] + 58.468;
   1:  PR[GP1:91,2] = PR[GP1:90,2] + -28.533;
   1:L PR[91] R[100]mm/sec CNT100;
   1:  PR[GP1:91,1] = PR[GP1:90,1] + 62.163;
   1:  PR[GP1:91,2] = PR[GP1:90,2] + -25.161;
   1:L PR[91] R[100]mm/sec CNT100;
   1:  PR[GP1:91,1] = PR[GP1:90,1] + 66.491;
   1:  PR[GP1:91,2] = PR[GP1:90,2] + -20.897;
   1:L PR[91] R[100]mm/sec CNT100;
   1:  PR[GP1:91,1] = PR[GP1:90,1] + 69.277;
   1:  PR[GP1:91,2] = PR[GP1:90,2] + -15.800;
   1:L PR[91] R[100]mm/sec CNT100;
   1:  PR[GP1:91,1] = PR[GP1:90,1] + 71.719;
   1:  PR[GP1:91,2] = PR[GP1:90,2] + -11.087;
   1:L PR[91] R[100]mm/sec CNT100;
   1:  PR[GP1:91,1] = PR[GP1:90,1] + 72.784;
   1:  PR[GP1:91,2] = PR[GP1:90,2] + -4.794;
   1:L PR[91] R[100]mm/sec CNT100;
   1:  PR[GP1:91,1] = PR[GP1:90,1] + 73.539;
   1:  PR[GP1:91,2] = PR[GP1:90,2] + -0.075;
   1:L PR[91] R[100]mm/sec CNT100;
   1:  PR[GP1:91,1] = PR[GP1:90,1] + 72.489;
   1:  PR[GP1:91,2] = PR[GP1:90,2] + 6.117;
   1:L PR[91] R[100]mm/sec CNT100;
   1:  PR[GP1:91,1] = PR[GP1:90,1] + 71.717;
   1:  PR[GP1:91,2] = PR[GP1:90,2] + 10.946;
   1:L PR[91] R[100]mm/sec CNT100;
   1:  PR[GP1:91,1] = PR[GP1:90,1] + 69.277;
   1:  PR[GP1:91,2] = PR[GP1:90,2] + 15.656;
   1:L PR[91] R[100]mm/sec CNT100;
   1:  PR[GP1:91,1] = PR[GP1:90,1] + 66.491;
   1:  PR[GP1:91,2] = PR[GP1:90,2] + 20.753;
   1:L PR[91] R[100]mm/sec CNT100;
   1:  PR[GP1:91,1] = PR[GP1:90,1] + 62.164;
   1:  PR[GP1:91,2] = PR[GP1:90,2] + 25.017;
   1:L PR[91] R[100]mm/sec CNT100;
   1:  PR[GP1:91,1] = PR[GP1:90,1] + 58.468;
   1:  PR[GP1:91,2] = PR[GP1:90,2] + 28.389;
   1:L PR[91] R[100]mm/sec CNT100;
   1:  PR[GP1:91,1] = PR[GP1:90,1] + 52.025;
   1:  PR[GP1:91,2] = PR[GP1:90,2] + 31.601;
   1:L PR[91] R[100]mm/sec CNT100;
   1:  PR[GP1:91,1] = PR[GP1:90,1] + 48.566;
   1:  PR[GP1:91,2] = PR[GP1:90,2] + 33.105;
   1:L PR[91] R[100]mm/sec CNT100;
   1:  PR[GP1:91,1] = PR[GP1:90,1] + 39.985;
   1:  PR[GP1:91,2] = PR[GP1:90,2] + 34.407;
   1:L PR[91] R[100]mm/sec CNT100;
   1:  PR[GP1:91,1] = PR[GP1:90,1] + 37.848;
   1:  PR[GP1:91,2] = PR[GP1:90,2] + 34.582;
   1:L PR[91] R[100]mm/sec CNT100;
   1:  PR[GP1:91,1] = PR[GP1:90,1] + 27.577;
   1:  PR[GP1:91,2] = PR[GP1:90,2] + 32.911;
   1:L PR[91] R[100]mm/sec CNT100;
   1:  PR[GP1:91,1] = PR[GP1:90,1] + 27.359;
   1:  PR[GP1:91,2] = PR[GP1:90,2] + 32.857;
   1:L PR[91] R[100]mm/sec CNT100;
   1:  PR[GP1:91,1] = PR[GP1:90,1] + 25.805;
   1:  PR[GP1:91,2] = PR[GP1:90,2] + 32.062;
   1:L PR[91] R[100]mm/sec CNT100;
   1:  PR[GP1:91,1] = PR[GP1:90,1] + 17.829;
   1:  PR[GP1:91,2] = PR[GP1:90,2] + 28.172;
   1:L PR[91] R[100]mm/sec CNT100;
   1:  PR[GP1:91,1] = PR[GP1:90,1] + 16.588;
   1:  PR[GP1:91,2] = PR[GP1:90,2] + 27.213;
   1:L PR[91] R[100]mm/sec CNT100;
   1:  PR[GP1:91,1] = PR[GP1:90,1] + 10.239;
   1:  PR[GP1:91,2] = PR[GP1:90,2] + 21.065;
   1:L PR[91] R[100]mm/sec CNT100;
   1:  PR[GP1:91,1] = PR[GP1:90,1] + 8.329;
   1:  PR[GP1:91,2] = PR[GP1:90,2] + 18.299;
   1:L PR[91] R[100]mm/sec CNT100;
   1:  PR[GP1:91,1] = PR[GP1:90,1] + 5.111;
   1:  PR[GP1:91,2] = PR[GP1:90,2] + 12.170;
   1:L PR[91] R[100]mm/sec CNT100;
   1:  PR[GP1:91,1] = PR[GP1:90,1] + 5.058;
   1:  PR[GP1:91,2] = PR[GP1:90,2] + 12.016;
   1:L PR[91] R[100]mm/sec CNT100;
   1:  PR[GP1:91,1] = PR[GP1:90,1] + 2.730;
   1:  PR[GP1:91,2] = PR[GP1:90,2] + 9.195;
   1:L PR[91] R[100]mm/sec CNT100;
   1:  PR[GP1:91,1] = PR[GP1:90,1] + 2.320;
   1:  PR[GP1:91,2] = PR[GP1:90,2] + 8.750;
   1:L PR[91] R[100]mm/sec CNT100;
   1:  PR[GP1:91,1] = PR[GP1:90,1] + 1.982;
   1:  PR[GP1:91,2] = PR[GP1:90,2] + 8.563;
   1:L PR[91] R[100]mm/sec CNT100;
   1:  PR[GP1:91,1] = PR[GP1:90,1] + -0.987;
   1:  PR[GP1:91,2] = PR[GP1:90,2] + 8.594;
   1:L PR[91] R[100]mm/sec CNT100;
   1:  ! -- Layer/Ebene 42 -- !;
   1:  PR[91] = PR[90];
   1:  PR[GP1:91,1] = PR[GP1:90,1] + -1.980;
   1:  PR[GP1:91,2] = PR[GP1:90,2] + 9.186;
   1:  PR[GP1:91,3] = PR[GP1:90,3] + 25.925;
   1:L PR[91] R[100]mm/sec CNT100;
   1:  PR[GP1:91,1] = PR[GP1:90,1] + -2.224;
   1:  PR[GP1:91,2] = PR[GP1:90,2] + 9.357;
   1:L PR[91] R[100]mm/sec CNT100;
   1:  PR[GP1:91,1] = PR[GP1:90,1] + -4.353;
   1:  PR[GP1:91,2] = PR[GP1:90,2] + 11.966;
   1:L PR[91] R[100]mm/sec CNT100;
   1:  PR[GP1:91,1] = PR[GP1:90,1] + -4.815;
   1:  PR[GP1:91,2] = PR[GP1:90,2] + 12.464;
   1:L PR[91] R[100]mm/sec CNT100;
   1:  PR[GP1:91,1] = PR[GP1:90,1] + -7.615;
   1:  PR[GP1:91,2] = PR[GP1:90,2] + 17.810;
   1:L PR[91] R[100]mm/sec CNT100;
   1:  PR[GP1:91,1] = PR[GP1:90,1] + -10.077;
   1:  PR[GP1:91,2] = PR[GP1:90,2] + 21.376;
   1:L PR[91] R[100]mm/sec CNT100;
   1:  PR[GP1:91,1] = PR[GP1:90,1] + -15.734;
   1:  PR[GP1:91,2] = PR[GP1:90,2] + 26.839;
   1:L PR[91] R[100]mm/sec CNT100;
   1:  PR[GP1:91,1] = PR[GP1:90,1] + -17.700;
   1:  PR[GP1:91,2] = PR[GP1:90,2] + 28.357;
   1:L PR[91] R[100]mm/sec CNT100;
   1:  PR[GP1:91,1] = PR[GP1:90,1] + -26.754;
   1:  PR[GP1:91,2] = PR[GP1:90,2] + 32.773;
   1:L PR[91] R[100]mm/sec CNT100;
   1:  PR[GP1:91,1] = PR[GP1:90,1] + -27.186;
   1:  PR[GP1:91,2] = PR[GP1:90,2] + 32.937;
   1:L PR[91] R[100]mm/sec CNT100;
   1:  PR[GP1:91,1] = PR[GP1:90,1] + -29.912;
   1:  PR[GP1:91,2] = PR[GP1:90,2] + 33.337;
   1:L PR[91] R[100]mm/sec CNT100;
   1:  PR[GP1:91,1] = PR[GP1:90,1] + -37.743;
   1:  PR[GP1:91,2] = PR[GP1:90,2] + 34.607;
   1:L PR[91] R[100]mm/sec CNT100;
   1:  PR[GP1:91,1] = PR[GP1:90,1] + -39.084;
   1:  PR[GP1:91,2] = PR[GP1:90,2] + 34.497;
   1:L PR[91] R[100]mm/sec CNT100;
   1:  PR[GP1:91,1] = PR[GP1:90,1] + -48.414;
   1:  PR[GP1:91,2] = PR[GP1:90,2] + 33.079;
   1:L PR[91] R[100]mm/sec CNT100;
   1:  PR[GP1:91,1] = PR[GP1:90,1] + -51.195;
   1:  PR[GP1:91,2] = PR[GP1:90,2] + 31.870;
   1:L PR[91] R[100]mm/sec CNT100;
   1:  PR[GP1:91,1] = PR[GP1:90,1] + -58.267;
   1:  PR[GP1:91,2] = PR[GP1:90,2] + 28.339;
   1:L PR[91] R[100]mm/sec CNT100;
   1:  PR[GP1:91,1] = PR[GP1:90,1] + -61.455;
   1:  PR[GP1:91,2] = PR[GP1:90,2] + 25.431;
   1:L PR[91] R[100]mm/sec CNT100;
   1:  PR[GP1:91,1] = PR[GP1:90,1] + -66.249;
   1:  PR[GP1:91,2] = PR[GP1:90,2] + 20.713;
   1:L PR[91] R[100]mm/sec CNT100;
   1:  PR[GP1:91,1] = PR[GP1:90,1] + -68.725;
   1:  PR[GP1:91,2] = PR[GP1:90,2] + 16.179;
   1:L PR[91] R[100]mm/sec CNT100;
   1:  PR[GP1:91,1] = PR[GP1:90,1] + -71.449;
   1:  PR[GP1:91,2] = PR[GP1:90,2] + 10.907;
   1:L PR[91] R[100]mm/sec CNT100;
   1:  PR[GP1:91,1] = PR[GP1:90,1] + -72.409;
   1:  PR[GP1:91,2] = PR[GP1:90,2] + 5.239;
   1:L PR[91] R[100]mm/sec CNT100;
   1:  PR[GP1:91,1] = PR[GP1:90,1] + -73.259;
   1:  PR[GP1:91,2] = PR[GP1:90,2] + -0.069;
   1:L PR[91] R[100]mm/sec CNT100;
   1:  PR[GP1:91,1] = PR[GP1:90,1] + -72.309;
   1:  PR[GP1:91,2] = PR[GP1:90,2] + -5.673;
   1:L PR[91] R[100]mm/sec CNT100;
   1:  PR[GP1:91,1] = PR[GP1:90,1] + -71.448;
   1:  PR[GP1:91,2] = PR[GP1:90,2] + -11.054;
   1:L PR[91] R[100]mm/sec CNT100;
   1:  PR[GP1:91,1] = PR[GP1:90,1] + -68.725;
   1:  PR[GP1:91,2] = PR[GP1:90,2] + -16.323;
   1:L PR[91] R[100]mm/sec CNT100;
   1:  PR[GP1:91,1] = PR[GP1:90,1] + -66.249;
   1:  PR[GP1:91,2] = PR[GP1:90,2] + -20.857;
   1:L PR[91] R[100]mm/sec CNT100;
   1:  PR[GP1:91,1] = PR[GP1:90,1] + -61.455;
   1:  PR[GP1:91,2] = PR[GP1:90,2] + -25.575;
   1:L PR[91] R[100]mm/sec CNT100;
   1:  PR[GP1:91,1] = PR[GP1:90,1] + -58.267;
   1:  PR[GP1:91,2] = PR[GP1:90,2] + -28.483;
   1:L PR[91] R[100]mm/sec CNT100;
   1:  PR[GP1:91,1] = PR[GP1:90,1] + -51.195;
   1:  PR[GP1:91,2] = PR[GP1:90,2] + -32.014;
   1:L PR[91] R[100]mm/sec CNT100;
   1:  PR[GP1:91,1] = PR[GP1:90,1] + -48.414;
   1:  PR[GP1:91,2] = PR[GP1:90,2] + -33.223;
   1:L PR[91] R[100]mm/sec CNT100;
   1:  PR[GP1:91,1] = PR[GP1:90,1] + -39.084;
   1:  PR[GP1:91,2] = PR[GP1:90,2] + -34.641;
   1:L PR[91] R[100]mm/sec CNT100;
   1:  PR[GP1:91,1] = PR[GP1:90,1] + -37.744;
   1:  PR[GP1:91,2] = PR[GP1:90,2] + -34.751;
   1:L PR[91] R[100]mm/sec CNT100;
   1:  PR[GP1:91,1] = PR[GP1:90,1] + -29.912;
   1:  PR[GP1:91,2] = PR[GP1:90,2] + -33.481;
   1:L PR[91] R[100]mm/sec CNT100;
   1:  PR[GP1:91,1] = PR[GP1:90,1] + -27.186;
   1:  PR[GP1:91,2] = PR[GP1:90,2] + -33.081;
   1:L PR[91] R[100]mm/sec CNT100;
   1:  PR[GP1:91,1] = PR[GP1:90,1] + -26.754;
   1:  PR[GP1:91,2] = PR[GP1:90,2] + -32.917;
   1:L PR[91] R[100]mm/sec CNT100;
   1:  PR[GP1:91,1] = PR[GP1:90,1] + -17.700;
   1:  PR[GP1:91,2] = PR[GP1:90,2] + -28.501;
   1:L PR[91] R[100]mm/sec CNT100;
   1:  PR[GP1:91,1] = PR[GP1:90,1] + -15.734;
   1:  PR[GP1:91,2] = PR[GP1:90,2] + -26.983;
   1:L PR[91] R[100]mm/sec CNT100;
   1:  PR[GP1:91,1] = PR[GP1:90,1] + -10.077;
   1:  PR[GP1:91,2] = PR[GP1:90,2] + -21.520;
   1:L PR[91] R[100]mm/sec CNT100;
   1:  PR[GP1:91,1] = PR[GP1:90,1] + -7.606;
   1:  PR[GP1:91,2] = PR[GP1:90,2] + -17.936;
   1:L PR[91] R[100]mm/sec CNT100;
   1:  PR[GP1:91,1] = PR[GP1:90,1] + -4.612;
   1:  PR[GP1:91,2] = PR[GP1:90,2] + -12.206;
   1:L PR[91] R[100]mm/sec CNT100;
   1:  PR[GP1:91,1] = PR[GP1:90,1] + -4.481;
   1:  PR[GP1:91,2] = PR[GP1:90,2] + -12.249;
   1:L PR[91] R[100]mm/sec CNT100;
   1:  PR[GP1:91,1] = PR[GP1:90,1] + -4.259;
   1:  PR[GP1:91,2] = PR[GP1:90,2] + -12.007;
   1:L PR[91] R[100]mm/sec CNT100;
   1:  PR[GP1:91,1] = PR[GP1:90,1] + -1.951;
   1:  PR[GP1:91,2] = PR[GP1:90,2] + -9.249;
   1:L PR[91] R[100]mm/sec CNT100;
   1:  PR[GP1:91,1] = PR[GP1:90,1] + -0.874;
   1:  PR[GP1:91,2] = PR[GP1:90,2] + -9.332;
   1:L PR[91] R[100]mm/sec CNT100;
   1:  PR[GP1:91,1] = PR[GP1:90,1] + -0.861;
   1:  PR[GP1:91,2] = PR[GP1:90,2] + -9.343;
   1:L PR[91] R[100]mm/sec CNT100;
   1:  PR[GP1:91,1] = PR[GP1:90,1] + 2.319;
   1:  PR[GP1:91,2] = PR[GP1:90,2] + -9.310;
   1:L PR[91] R[100]mm/sec CNT100;
   1:  PR[GP1:91,1] = PR[GP1:90,1] + 2.734;
   1:  PR[GP1:91,2] = PR[GP1:90,2] + -10.100;
   1:L PR[91] R[100]mm/sec CNT100;
   1:  PR[GP1:91,1] = PR[GP1:90,1] + 3.143;
   1:  PR[GP1:91,2] = PR[GP1:90,2] + -10.571;
   1:L PR[91] R[100]mm/sec CNT100;
   1:  PR[GP1:91,1] = PR[GP1:90,1] + 4.455;
   1:  PR[GP1:91,2] = PR[GP1:90,2] + -12.000;
   1:L PR[91] R[100]mm/sec CNT100;
   1:  PR[GP1:91,1] = PR[GP1:90,1] + 4.813;
   1:  PR[GP1:91,2] = PR[GP1:90,2] + -12.428;
   1:L PR[91] R[100]mm/sec CNT100;
   1:  PR[GP1:91,1] = PR[GP1:90,1] + 4.983;
   1:  PR[GP1:91,2] = PR[GP1:90,2] + -12.536;
   1:L PR[91] R[100]mm/sec CNT100;
   1:  PR[GP1:91,1] = PR[GP1:90,1] + 7.809;
   1:  PR[GP1:91,2] = PR[GP1:90,2] + -17.914;
   1:L PR[91] R[100]mm/sec CNT100;
   1:  PR[GP1:91,1] = PR[GP1:90,1] + 10.284;
   1:  PR[GP1:91,2] = PR[GP1:90,2] + -21.503;
   1:L PR[91] R[100]mm/sec CNT100;
   1:  PR[GP1:91,1] = PR[GP1:90,1] + 15.937;
   1:  PR[GP1:91,2] = PR[GP1:90,2] + -26.977;
   1:L PR[91] R[100]mm/sec CNT100;
   1:  PR[GP1:91,1] = PR[GP1:90,1] + 17.903;
   1:  PR[GP1:91,2] = PR[GP1:90,2] + -28.497;
   1:L PR[91] R[100]mm/sec CNT100;
   1:  PR[GP1:91,1] = PR[GP1:90,1] + 26.953;
   1:  PR[GP1:91,2] = PR[GP1:90,2] + -32.910;
   1:L PR[91] R[100]mm/sec CNT100;
   1:  PR[GP1:91,1] = PR[GP1:90,1] + 27.388;
   1:  PR[GP1:91,2] = PR[GP1:90,2] + -33.075;
   1:L PR[91] R[100]mm/sec CNT100;
   1:  PR[GP1:91,1] = PR[GP1:90,1] + 30.126;
   1:  PR[GP1:91,2] = PR[GP1:90,2] + -33.478;
   1:L PR[91] R[100]mm/sec CNT100;
   1:  PR[GP1:91,1] = PR[GP1:90,1] + 37.947;
   1:  PR[GP1:91,2] = PR[GP1:90,2] + -34.751;
   1:L PR[91] R[100]mm/sec CNT100;
   1:  PR[GP1:91,1] = PR[GP1:90,1] + 39.285;
   1:  PR[GP1:91,2] = PR[GP1:90,2] + -34.641;
   1:L PR[91] R[100]mm/sec CNT100;
   1:  PR[GP1:91,1] = PR[GP1:90,1] + 48.620;
   1:  PR[GP1:91,2] = PR[GP1:90,2] + -33.224;
   1:L PR[91] R[100]mm/sec CNT100;
   1:  PR[GP1:91,1] = PR[GP1:90,1] + 51.401;
   1:  PR[GP1:91,2] = PR[GP1:90,2] + -32.016;
   1:L PR[91] R[100]mm/sec CNT100;
   1:  PR[GP1:91,1] = PR[GP1:90,1] + 58.476;
   1:  PR[GP1:91,2] = PR[GP1:90,2] + -28.488;
   1:L PR[91] R[100]mm/sec CNT100;
   1:  PR[GP1:91,1] = PR[GP1:90,1] + 61.664;
   1:  PR[GP1:91,2] = PR[GP1:90,2] + -25.580;
   1:L PR[91] R[100]mm/sec CNT100;
   1:  PR[GP1:91,1] = PR[GP1:90,1] + 66.460;
   1:  PR[GP1:91,2] = PR[GP1:90,2] + -20.853;
   1:L PR[91] R[100]mm/sec CNT100;
   1:  PR[GP1:91,1] = PR[GP1:90,1] + 68.936;
   1:  PR[GP1:91,2] = PR[GP1:90,2] + -16.322;
   1:L PR[91] R[100]mm/sec CNT100;
   1:  PR[GP1:91,1] = PR[GP1:90,1] + 71.662;
   1:  PR[GP1:91,2] = PR[GP1:90,2] + -11.062;
   1:L PR[91] R[100]mm/sec CNT100;
   1:  PR[GP1:91,1] = PR[GP1:90,1] + 72.621;
   1:  PR[GP1:91,2] = PR[GP1:90,2] + -5.392;
   1:L PR[91] R[100]mm/sec CNT100;
   1:  PR[GP1:91,1] = PR[GP1:90,1] + 73.473;
   1:  PR[GP1:91,2] = PR[GP1:90,2] + -0.075;
   1:L PR[91] R[100]mm/sec CNT100;
   1:  PR[GP1:91,1] = PR[GP1:90,1] + 72.522;
   1:  PR[GP1:91,2] = PR[GP1:90,2] + 5.531;
   1:L PR[91] R[100]mm/sec CNT100;
   1:  PR[GP1:91,1] = PR[GP1:90,1] + 71.661;
   1:  PR[GP1:91,2] = PR[GP1:90,2] + 10.921;
   1:L PR[91] R[100]mm/sec CNT100;
   1:  PR[GP1:91,1] = PR[GP1:90,1] + 68.936;
   1:  PR[GP1:91,2] = PR[GP1:90,2] + 16.178;
   1:L PR[91] R[100]mm/sec CNT100;
   1:  PR[GP1:91,1] = PR[GP1:90,1] + 66.460;
   1:  PR[GP1:91,2] = PR[GP1:90,2] + 20.709;
   1:L PR[91] R[100]mm/sec CNT100;
   1:  PR[GP1:91,1] = PR[GP1:90,1] + 61.664;
   1:  PR[GP1:91,2] = PR[GP1:90,2] + 25.436;
   1:L PR[91] R[100]mm/sec CNT100;
   1:  PR[GP1:91,1] = PR[GP1:90,1] + 58.476;
   1:  PR[GP1:91,2] = PR[GP1:90,2] + 28.344;
   1:L PR[91] R[100]mm/sec CNT100;
   1:  PR[GP1:91,1] = PR[GP1:90,1] + 51.401;
   1:  PR[GP1:91,2] = PR[GP1:90,2] + 31.872;
   1:L PR[91] R[100]mm/sec CNT100;
   1:  PR[GP1:91,1] = PR[GP1:90,1] + 48.620;
   1:  PR[GP1:91,2] = PR[GP1:90,2] + 33.080;
   1:L PR[91] R[100]mm/sec CNT100;
   1:  PR[GP1:91,1] = PR[GP1:90,1] + 39.285;
   1:  PR[GP1:91,2] = PR[GP1:90,2] + 34.497;
   1:L PR[91] R[100]mm/sec CNT100;
   1:  PR[GP1:91,1] = PR[GP1:90,1] + 37.947;
   1:  PR[GP1:91,2] = PR[GP1:90,2] + 34.607;
   1:L PR[91] R[100]mm/sec CNT100;
   1:  PR[GP1:91,1] = PR[GP1:90,1] + 30.126;
   1:  PR[GP1:91,2] = PR[GP1:90,2] + 33.334;
   1:L PR[91] R[100]mm/sec CNT100;
   1:  PR[GP1:91,1] = PR[GP1:90,1] + 27.387;
   1:  PR[GP1:91,2] = PR[GP1:90,2] + 32.931;
   1:L PR[91] R[100]mm/sec CNT100;
   1:  PR[GP1:91,1] = PR[GP1:90,1] + 26.952;
   1:  PR[GP1:91,2] = PR[GP1:90,2] + 32.766;
   1:L PR[91] R[100]mm/sec CNT100;
   1:  PR[GP1:91,1] = PR[GP1:90,1] + 17.903;
   1:  PR[GP1:91,2] = PR[GP1:90,2] + 28.353;
   1:L PR[91] R[100]mm/sec CNT100;
   1:  PR[GP1:91,1] = PR[GP1:90,1] + 15.937;
   1:  PR[GP1:91,2] = PR[GP1:90,2] + 26.833;
   1:L PR[91] R[100]mm/sec CNT100;
   1:  PR[GP1:91,1] = PR[GP1:90,1] + 10.284;
   1:  PR[GP1:91,2] = PR[GP1:90,2] + 21.359;
   1:L PR[91] R[100]mm/sec CNT100;
   1:  PR[GP1:91,1] = PR[GP1:90,1] + 7.819;
   1:  PR[GP1:91,2] = PR[GP1:90,2] + 17.788;
   1:L PR[91] R[100]mm/sec CNT100;
   1:  PR[GP1:91,1] = PR[GP1:90,1] + 5.021;
   1:  PR[GP1:91,2] = PR[GP1:90,2] + 12.464;
   1:L PR[91] R[100]mm/sec CNT100;
   1:  PR[GP1:91,1] = PR[GP1:90,1] + 4.549;
   1:  PR[GP1:91,2] = PR[GP1:90,2] + 11.958;
   1:L PR[91] R[100]mm/sec CNT100;
   1:  PR[GP1:91,1] = PR[GP1:90,1] + 2.606;
   1:  PR[GP1:91,2] = PR[GP1:90,2] + 9.604;
   1:L PR[91] R[100]mm/sec CNT100;
   1:  PR[GP1:91,1] = PR[GP1:90,1] + 2.292;
   1:  PR[GP1:91,2] = PR[GP1:90,2] + 9.263;
   1:L PR[91] R[100]mm/sec CNT100;
   1:  PR[GP1:91,1] = PR[GP1:90,1] + 1.987;
   1:  PR[GP1:91,2] = PR[GP1:90,2] + 9.094;
   1:L PR[91] R[100]mm/sec CNT100;
   1:  PR[GP1:91,1] = PR[GP1:90,1] + -1.205;
   1:  PR[GP1:91,2] = PR[GP1:90,2] + 9.128;
   1:L PR[91] R[100]mm/sec CNT100;
   1:  ! -- Layer/Ebene 43 -- !;
   1:  PR[91] = PR[90];
   1:  PR[GP1:91,1] = PR[GP1:90,1] + -1.957;
   1:  PR[GP1:91,2] = PR[GP1:90,2] + 9.701;
   1:  PR[GP1:91,3] = PR[GP1:90,3] + 26.535;
   1:L PR[91] R[100]mm/sec CNT100;
   1:  PR[GP1:91,1] = PR[GP1:90,1] + -2.184;
   1:  PR[GP1:91,2] = PR[GP1:90,2] + 9.861;
   1:L PR[91] R[100]mm/sec CNT100;
   1:  PR[GP1:91,1] = PR[GP1:90,1] + -3.464;
   1:  PR[GP1:91,2] = PR[GP1:90,2] + 11.428;
   1:L PR[91] R[100]mm/sec CNT100;
   1:  PR[GP1:91,1] = PR[GP1:90,1] + -4.781;
   1:  PR[GP1:91,2] = PR[GP1:90,2] + 12.849;
   1:L PR[91] R[100]mm/sec CNT100;
   1:  PR[GP1:91,1] = PR[GP1:90,1] + -7.104;
   1:  PR[GP1:91,2] = PR[GP1:90,2] + 17.298;
   1:L PR[91] R[100]mm/sec CNT100;
   1:  PR[GP1:91,1] = PR[GP1:90,1] + -10.121;
   1:  PR[GP1:91,2] = PR[GP1:90,2] + 21.668;
   1:L PR[91] R[100]mm/sec CNT100;
   1:  PR[GP1:91,1] = PR[GP1:90,1] + -15.082;
   1:  PR[GP1:91,2] = PR[GP1:90,2] + 26.459;
   1:L PR[91] R[100]mm/sec CNT100;
   1:  PR[GP1:91,1] = PR[GP1:90,1] + -17.773;
   1:  PR[GP1:91,2] = PR[GP1:90,2] + 28.537;
   1:L PR[91] R[100]mm/sec CNT100;
   1:  PR[GP1:91,1] = PR[GP1:90,1] + -25.993;
   1:  PR[GP1:91,2] = PR[GP1:90,2] + 32.546;
   1:L PR[91] R[100]mm/sec CNT100;
   1:  PR[GP1:91,1] = PR[GP1:90,1] + -27.252;
   1:  PR[GP1:91,2] = PR[GP1:90,2] + 33.024;
   1:L PR[91] R[100]mm/sec CNT100;
   1:  PR[GP1:91,1] = PR[GP1:90,1] + -34.407;
   1:  PR[GP1:91,2] = PR[GP1:90,2] + 34.074;
   1:L PR[91] R[100]mm/sec CNT100;
   1:  PR[GP1:91,1] = PR[GP1:90,1] + -37.843;
   1:  PR[GP1:91,2] = PR[GP1:90,2] + 34.631;
   1:L PR[91] R[100]mm/sec CNT100;
   1:  PR[GP1:91,1] = PR[GP1:90,1] + -38.385;
   1:  PR[GP1:91,2] = PR[GP1:90,2] + 34.586;
   1:L PR[91] R[100]mm/sec CNT100;
   1:  PR[GP1:91,1] = PR[GP1:90,1] + -48.469;
   1:  PR[GP1:91,2] = PR[GP1:90,2] + 33.055;
   1:L PR[91] R[100]mm/sec CNT100;
   1:  PR[GP1:91,1] = PR[GP1:90,1] + -50.572;
   1:  PR[GP1:91,2] = PR[GP1:90,2] + 32.141;
   1:L PR[91] R[100]mm/sec CNT100;
   1:  PR[GP1:91,1] = PR[GP1:90,1] + -58.275;
   1:  PR[GP1:91,2] = PR[GP1:90,2] + 28.293;
   1:L PR[91] R[100]mm/sec CNT100;
   1:  PR[GP1:91,1] = PR[GP1:90,1] + -60.956;
   1:  PR[GP1:91,2] = PR[GP1:90,2] + 25.849;
   1:L PR[91] R[100]mm/sec CNT100;
   1:  PR[GP1:91,1] = PR[GP1:90,1] + -66.218;
   1:  PR[GP1:91,2] = PR[GP1:90,2] + 20.670;
   1:L PR[91] R[100]mm/sec CNT100;
   1:  PR[GP1:91,1] = PR[GP1:90,1] + -68.384;
   1:  PR[GP1:91,2] = PR[GP1:90,2] + 16.702;
   1:L PR[91] R[100]mm/sec CNT100;
   1:  PR[GP1:91,1] = PR[GP1:90,1] + -71.392;
   1:  PR[GP1:91,2] = PR[GP1:90,2] + 10.882;
   1:L PR[91] R[100]mm/sec CNT100;
   1:  PR[GP1:91,1] = PR[GP1:90,1] + -72.247;
   1:  PR[GP1:91,2] = PR[GP1:90,2] + 5.835;
   1:L PR[91] R[100]mm/sec CNT100;
   1:  PR[GP1:91,1] = PR[GP1:90,1] + -73.193;
   1:  PR[GP1:91,2] = PR[GP1:90,2] + -0.069;
   1:L PR[91] R[100]mm/sec CNT100;
   1:  PR[GP1:91,1] = PR[GP1:90,1] + -72.342;
   1:  PR[GP1:91,2] = PR[GP1:90,2] + -5.088;
   1:L PR[91] R[100]mm/sec CNT100;
   1:  PR[GP1:91,1] = PR[GP1:90,1] + -71.391;
   1:  PR[GP1:91,2] = PR[GP1:90,2] + -11.028;
   1:L PR[91] R[100]mm/sec CNT100;
   1:  PR[GP1:91,1] = PR[GP1:90,1] + -68.384;
   1:  PR[GP1:91,2] = PR[GP1:90,2] + -16.846;
   1:L PR[91] R[100]mm/sec CNT100;
   1:  PR[GP1:91,1] = PR[GP1:90,1] + -66.218;
   1:  PR[GP1:91,2] = PR[GP1:90,2] + -20.814;
   1:L PR[91] R[100]mm/sec CNT100;
   1:  PR[GP1:91,1] = PR[GP1:90,1] + -60.956;
   1:  PR[GP1:91,2] = PR[GP1:90,2] + -25.993;
   1:L PR[91] R[100]mm/sec CNT100;
   1:  PR[GP1:91,1] = PR[GP1:90,1] + -58.275;
   1:  PR[GP1:91,2] = PR[GP1:90,2] + -28.437;
   1:L PR[91] R[100]mm/sec CNT100;
   1:  PR[GP1:91,1] = PR[GP1:90,1] + -50.572;
   1:  PR[GP1:91,2] = PR[GP1:90,2] + -32.285;
   1:L PR[91] R[100]mm/sec CNT100;
   1:  PR[GP1:91,1] = PR[GP1:90,1] + -48.469;
   1:  PR[GP1:91,2] = PR[GP1:90,2] + -33.199;
   1:L PR[91] R[100]mm/sec CNT100;
   1:  PR[GP1:91,1] = PR[GP1:90,1] + -38.386;
   1:  PR[GP1:91,2] = PR[GP1:90,2] + -34.730;
   1:L PR[91] R[100]mm/sec CNT100;
   1:  PR[GP1:91,1] = PR[GP1:90,1] + -37.843;
   1:  PR[GP1:91,2] = PR[GP1:90,2] + -34.775;
   1:L PR[91] R[100]mm/sec CNT100;
   1:  PR[GP1:91,1] = PR[GP1:90,1] + -34.407;
   1:  PR[GP1:91,2] = PR[GP1:90,2] + -34.218;
   1:L PR[91] R[100]mm/sec CNT100;
   1:  PR[GP1:91,1] = PR[GP1:90,1] + -27.252;
   1:  PR[GP1:91,2] = PR[GP1:90,2] + -33.169;
   1:L PR[91] R[100]mm/sec CNT100;
   1:  PR[GP1:91,1] = PR[GP1:90,1] + -25.993;
   1:  PR[GP1:91,2] = PR[GP1:90,2] + -32.690;
   1:L PR[91] R[100]mm/sec CNT100;
   1:  PR[GP1:91,1] = PR[GP1:90,1] + -17.773;
   1:  PR[GP1:91,2] = PR[GP1:90,2] + -28.681;
   1:L PR[91] R[100]mm/sec CNT100;
   1:  PR[GP1:91,1] = PR[GP1:90,1] + -15.082;
   1:  PR[GP1:91,2] = PR[GP1:90,2] + -26.603;
   1:L PR[91] R[100]mm/sec CNT100;
   1:  PR[GP1:91,1] = PR[GP1:90,1] + -10.121;
   1:  PR[GP1:91,2] = PR[GP1:90,2] + -21.812;
   1:L PR[91] R[100]mm/sec CNT100;
   1:  PR[GP1:91,1] = PR[GP1:90,1] + -7.092;
   1:  PR[GP1:91,2] = PR[GP1:90,2] + -17.420;
   1:L PR[91] R[100]mm/sec CNT100;
   1:  PR[GP1:91,1] = PR[GP1:90,1] + -4.580;
   1:  PR[GP1:91,2] = PR[GP1:90,2] + -12.611;
   1:L PR[91] R[100]mm/sec CNT100;
   1:  PR[GP1:91,1] = PR[GP1:90,1] + -4.452;
   1:  PR[GP1:91,2] = PR[GP1:90,2] + -12.654;
   1:L PR[91] R[100]mm/sec CNT100;
   1:  PR[GP1:91,1] = PR[GP1:90,1] + -3.407;
   1:  PR[GP1:91,2] = PR[GP1:90,2] + -11.510;
   1:L PR[91] R[100]mm/sec CNT100;
   1:  PR[GP1:91,1] = PR[GP1:90,1] + -1.961;
   1:  PR[GP1:91,2] = PR[GP1:90,2] + -9.783;
   1:L PR[91] R[100]mm/sec CNT100;
   1:  PR[GP1:91,1] = PR[GP1:90,1] + -1.134;
   1:  PR[GP1:91,2] = PR[GP1:90,2] + -9.846;
   1:L PR[91] R[100]mm/sec CNT100;
   1:  PR[GP1:91,1] = PR[GP1:90,1] + 2.273;
   1:  PR[GP1:91,2] = PR[GP1:90,2] + -9.811;
   1:L PR[91] R[100]mm/sec CNT100;
   1:  PR[GP1:91,1] = PR[GP1:90,1] + 2.577;
   1:  PR[GP1:91,2] = PR[GP1:90,2] + -10.386;
   1:L PR[91] R[100]mm/sec CNT100;
   1:  PR[GP1:91,1] = PR[GP1:90,1] + 3.589;
   1:  PR[GP1:91,2] = PR[GP1:90,2] + -11.504;
   1:L PR[91] R[100]mm/sec CNT100;
   1:  PR[GP1:91,1] = PR[GP1:90,1] + 4.599;
   1:  PR[GP1:91,2] = PR[GP1:90,2] + -12.714;
   1:L PR[91] R[100]mm/sec CNT100;
   1:  PR[GP1:91,1] = PR[GP1:90,1] + 4.951;
   1:  PR[GP1:91,2] = PR[GP1:90,2] + -12.936;
   1:L PR[91] R[100]mm/sec CNT100;
   1:  PR[GP1:91,1] = PR[GP1:90,1] + 7.296;
   1:  PR[GP1:91,2] = PR[GP1:90,2] + -17.399;
   1:L PR[91] R[100]mm/sec CNT100;
   1:  PR[GP1:91,1] = PR[GP1:90,1] + 10.329;
   1:  PR[GP1:91,2] = PR[GP1:90,2] + -21.797;
   1:L PR[91] R[100]mm/sec CNT100;
   1:  PR[GP1:91,1] = PR[GP1:90,1] + 15.286;
   1:  PR[GP1:91,2] = PR[GP1:90,2] + -26.597;
   1:L PR[91] R[100]mm/sec CNT100;
   1:  PR[GP1:91,1] = PR[GP1:90,1] + 17.978;
   1:  PR[GP1:91,2] = PR[GP1:90,2] + -28.678;
   1:L PR[91] R[100]mm/sec CNT100;
   1:  PR[GP1:91,1] = PR[GP1:90,1] + 26.193;
   1:  PR[GP1:91,2] = PR[GP1:90,2] + -32.684;
   1:L PR[91] R[100]mm/sec CNT100;
   1:  PR[GP1:91,1] = PR[GP1:90,1] + 27.454;
   1:  PR[GP1:91,2] = PR[GP1:90,2] + -33.163;
   1:L PR[91] R[100]mm/sec CNT100;
   1:  PR[GP1:91,1] = PR[GP1:90,1] + 34.621;
   1:  PR[GP1:91,2] = PR[GP1:90,2] + -34.218;
   1:L PR[91] R[100]mm/sec CNT100;
   1:  PR[GP1:91,1] = PR[GP1:90,1] + 38.046;
   1:  PR[GP1:91,2] = PR[GP1:90,2] + -34.775;
   1:L PR[91] R[100]mm/sec CNT100;
   1:  PR[GP1:91,1] = PR[GP1:90,1] + 38.586;
   1:  PR[GP1:91,2] = PR[GP1:90,2] + -34.731;
   1:L PR[91] R[100]mm/sec CNT100;
   1:  PR[GP1:91,1] = PR[GP1:90,1] + 48.675;
   1:  PR[GP1:91,2] = PR[GP1:90,2] + -33.199;
   1:L PR[91] R[100]mm/sec CNT100;
   1:  PR[GP1:91,1] = PR[GP1:90,1] + 50.777;
   1:  PR[GP1:91,2] = PR[GP1:90,2] + -32.286;
   1:L PR[91] R[100]mm/sec CNT100;
   1:  PR[GP1:91,1] = PR[GP1:90,1] + 58.484;
   1:  PR[GP1:91,2] = PR[GP1:90,2] + -28.443;
   1:L PR[91] R[100]mm/sec CNT100;
   1:  PR[GP1:91,1] = PR[GP1:90,1] + 61.164;
   1:  PR[GP1:91,2] = PR[GP1:90,2] + -25.998;
   1:L PR[91] R[100]mm/sec CNT100;
   1:  PR[GP1:91,1] = PR[GP1:90,1] + 66.429;
   1:  PR[GP1:91,2] = PR[GP1:90,2] + -20.810;
   1:L PR[91] R[100]mm/sec CNT100;
   1:  PR[GP1:91,1] = PR[GP1:90,1] + 68.596;
   1:  PR[GP1:91,2] = PR[GP1:90,2] + -16.844;
   1:L PR[91] R[100]mm/sec CNT100;
   1:  PR[GP1:91,1] = PR[GP1:90,1] + 71.605;
   1:  PR[GP1:91,2] = PR[GP1:90,2] + -11.038;
   1:L PR[91] R[100]mm/sec CNT100;
   1:  PR[GP1:91,1] = PR[GP1:90,1] + 72.459;
   1:  PR[GP1:91,2] = PR[GP1:90,2] + -5.989;
   1:L PR[91] R[100]mm/sec CNT100;
   1:  PR[GP1:91,1] = PR[GP1:90,1] + 73.406;
   1:  PR[GP1:91,2] = PR[GP1:90,2] + -0.075;
   1:L PR[91] R[100]mm/sec CNT100;
   1:  PR[GP1:91,1] = PR[GP1:90,1] + 72.555;
   1:  PR[GP1:91,2] = PR[GP1:90,2] + 4.946;
   1:L PR[91] R[100]mm/sec CNT100;
   1:  PR[GP1:91,1] = PR[GP1:90,1] + 71.604;
   1:  PR[GP1:91,2] = PR[GP1:90,2] + 10.896;
   1:L PR[91] R[100]mm/sec CNT100;
   1:  PR[GP1:91,1] = PR[GP1:90,1] + 68.596;
   1:  PR[GP1:91,2] = PR[GP1:90,2] + 16.701;
   1:L PR[91] R[100]mm/sec CNT100;
   1:  PR[GP1:91,1] = PR[GP1:90,1] + 66.429;
   1:  PR[GP1:91,2] = PR[GP1:90,2] + 20.666;
   1:L PR[91] R[100]mm/sec CNT100;
   1:  PR[GP1:91,1] = PR[GP1:90,1] + 61.164;
   1:  PR[GP1:91,2] = PR[GP1:90,2] + 25.854;
   1:L PR[91] R[100]mm/sec CNT100;
   1:  PR[GP1:91,1] = PR[GP1:90,1] + 58.484;
   1:  PR[GP1:91,2] = PR[GP1:90,2] + 28.299;
   1:L PR[91] R[100]mm/sec CNT100;
   1:  PR[GP1:91,1] = PR[GP1:90,1] + 50.777;
   1:  PR[GP1:91,2] = PR[GP1:90,2] + 32.142;
   1:L PR[91] R[100]mm/sec CNT100;
   1:  PR[GP1:91,1] = PR[GP1:90,1] + 48.675;
   1:  PR[GP1:91,2] = PR[GP1:90,2] + 33.055;
   1:L PR[91] R[100]mm/sec CNT100;
   1:  PR[GP1:91,1] = PR[GP1:90,1] + 38.586;
   1:  PR[GP1:91,2] = PR[GP1:90,2] + 34.587;
   1:L PR[91] R[100]mm/sec CNT100;
   1:  PR[GP1:91,1] = PR[GP1:90,1] + 38.046;
   1:  PR[GP1:91,2] = PR[GP1:90,2] + 34.631;
   1:L PR[91] R[100]mm/sec CNT100;
   1:  PR[GP1:91,1] = PR[GP1:90,1] + 34.621;
   1:  PR[GP1:91,2] = PR[GP1:90,2] + 34.074;
   1:L PR[91] R[100]mm/sec CNT100;
   1:  PR[GP1:91,1] = PR[GP1:90,1] + 27.454;
   1:  PR[GP1:91,2] = PR[GP1:90,2] + 33.019;
   1:L PR[91] R[100]mm/sec CNT100;
   1:  PR[GP1:91,1] = PR[GP1:90,1] + 26.193;
   1:  PR[GP1:91,2] = PR[GP1:90,2] + 32.540;
   1:L PR[91] R[100]mm/sec CNT100;
   1:  PR[GP1:91,1] = PR[GP1:90,1] + 17.977;
   1:  PR[GP1:91,2] = PR[GP1:90,2] + 28.534;
   1:L PR[91] R[100]mm/sec CNT100;
   1:  PR[GP1:91,1] = PR[GP1:90,1] + 15.286;
   1:  PR[GP1:91,2] = PR[GP1:90,2] + 26.453;
   1:L PR[91] R[100]mm/sec CNT100;
   1:  PR[GP1:91,1] = PR[GP1:90,1] + 10.329;
   1:  PR[GP1:91,2] = PR[GP1:90,2] + 21.653;
   1:L PR[91] R[100]mm/sec CNT100;
   1:  PR[GP1:91,1] = PR[GP1:90,1] + 7.308;
   1:  PR[GP1:91,2] = PR[GP1:90,2] + 17.278;
   1:L PR[91] R[100]mm/sec CNT100;
   1:  PR[GP1:91,1] = PR[GP1:90,1] + 4.988;
   1:  PR[GP1:91,2] = PR[GP1:90,2] + 12.864;
   1:L PR[91] R[100]mm/sec CNT100;
   1:  PR[GP1:91,1] = PR[GP1:90,1] + 3.644;
   1:  PR[GP1:91,2] = PR[GP1:90,2] + 11.419;
   1:L PR[91] R[100]mm/sec CNT100;
   1:  PR[GP1:91,1] = PR[GP1:90,1] + 2.483;
   1:  PR[GP1:91,2] = PR[GP1:90,2] + 10.013;
   1:L PR[91] R[100]mm/sec CNT100;
   1:  PR[GP1:91,1] = PR[GP1:90,1] + 2.264;
   1:  PR[GP1:91,2] = PR[GP1:90,2] + 9.775;
   1:L PR[91] R[100]mm/sec CNT100;
   1:  PR[GP1:91,1] = PR[GP1:90,1] + 1.992;
   1:  PR[GP1:91,2] = PR[GP1:90,2] + 9.625;
   1:L PR[91] R[100]mm/sec CNT100;
   1:  PR[GP1:91,1] = PR[GP1:90,1] + -1.422;
   1:  PR[GP1:91,2] = PR[GP1:90,2] + 9.661;
   1:L PR[91] R[100]mm/sec CNT100;
   1:  ! -- Layer/Ebene 44 -- !;
   1:  PR[91] = PR[90];
   1:  PR[GP1:91,1] = PR[GP1:90,1] + -2.043;
   1:  PR[GP1:91,2] = PR[GP1:90,2] + 10.240;
   1:  PR[GP1:91,3] = PR[GP1:90,3] + 27.145;
   1:L PR[91] R[100]mm/sec CNT100;
   1:  PR[GP1:91,1] = PR[GP1:90,1] + -2.574;
   1:  PR[GP1:91,2] = PR[GP1:90,2] + 10.890;
   1:L PR[91] R[100]mm/sec CNT100;
   1:  PR[GP1:91,1] = PR[GP1:90,1] + -4.826;
   1:  PR[GP1:91,2] = PR[GP1:90,2] + 13.319;
   1:L PR[91] R[100]mm/sec CNT100;
   1:  PR[GP1:91,1] = PR[GP1:90,1] + -4.840;
   1:  PR[GP1:91,2] = PR[GP1:90,2] + 13.443;
   1:L PR[91] R[100]mm/sec CNT100;
   1:  PR[GP1:91,1] = PR[GP1:90,1] + -6.593;
   1:  PR[GP1:91,2] = PR[GP1:90,2] + 16.786;
   1:L PR[91] R[100]mm/sec CNT100;
   1:  PR[GP1:91,1] = PR[GP1:90,1] + -10.165;
   1:  PR[GP1:91,2] = PR[GP1:90,2] + 21.960;
   1:L PR[91] R[100]mm/sec CNT100;
   1:  PR[GP1:91,1] = PR[GP1:90,1] + -14.429;
   1:  PR[GP1:91,2] = PR[GP1:90,2] + 26.078;
   1:L PR[91] R[100]mm/sec CNT100;
   1:  PR[GP1:91,1] = PR[GP1:90,1] + -17.846;
   1:  PR[GP1:91,2] = PR[GP1:90,2] + 28.717;
   1:L PR[91] R[100]mm/sec CNT100;
   1:  PR[GP1:91,1] = PR[GP1:90,1] + -25.233;
   1:  PR[GP1:91,2] = PR[GP1:90,2] + 32.319;
   1:L PR[91] R[100]mm/sec CNT100;
   1:  PR[GP1:91,1] = PR[GP1:90,1] + -27.317;
   1:  PR[GP1:91,2] = PR[GP1:90,2] + 33.112;
   1:L PR[91] R[100]mm/sec CNT100;
   1:  PR[GP1:91,1] = PR[GP1:90,1] + -37.801;
   1:  PR[GP1:91,2] = PR[GP1:90,2] + 34.649;
   1:L PR[91] R[100]mm/sec CNT100;
   1:  PR[GP1:91,1] = PR[GP1:90,1] + -37.881;
   1:  PR[GP1:91,2] = PR[GP1:90,2] + 34.655;
   1:L PR[91] R[100]mm/sec CNT100;
